(* CODESYS project comlibv2_gd.library
   Company: G.D Spa
   Version: 1.0.0.3
   Placeholder: COMlibV2_GD
   Title: COMlibV2_GD

Project tree, tasks and I/O mapping:
  libraries: Tc2_Standard, * (Beckhoff Automation GmbH); Tc2_System, * (Beckhoff Automation GmbH); Tc3_Module, * (Beckhoff Automation GmbH)
  Data types/
    COMlibV2/
      [Internal]/
        AdsSerialComm/
          data type ComADSSerialConfig_1
          data type ComADSServerCmd
        data type ComDebugBuffer
      AdsSerialComm/
        data type ComDTRCtrl_t
        data type ComRTSCtrl_t
        data type ComSerialConfig
        data type ComStopBits_t
      Hardware Types/
        data type EL6inData22B
        data type EL6outData22B
        data type IE6inData11B
        data type IE6outData11B
        data type KL6inData
        data type KL6inData22B
        data type KL6inData5B
        data type KL6outData
        data type KL6outData22B
        data type KL6outData5B
        data type M8000inData
        data type M8000outData
        data type PcComInData
        data type PcComOutData
      data type ComBuffer
      data type ComError_t
      data type ComHandshake_t
      data type ComParity_t
      data type ComRegisterData_t
      data type ComRegisterList_t
      data type ComSerialLineMode_t
  Global Variables/
    global variables Global_Constants
    global variables Global_Constants_ComLibVersion
    global variables Global_Variables
    global variables Variable_Configuration
  POUs/
    COMlibV2/
      [Internal]/
        function block _ReceiveString [ST]
        function block _SendString [ST]
        function _strncpy [ST]
      Background Communication/
        function block SerialLineControl [ST]
        function block SerialLineControlADS [ST]
        function block SerialLineControlM8000 [ST]
      CO_Nfiguration/
        function block KL6configuration [ST]
        function block KL6ReadRegisters [ST]
        function block KL6WriteRegisters [ST]
        function block M8000configuration [ST]
      Send + Receive/
        function block ReceiveByte [ST]
        function block ReceiveData [ST]
        function block ReceiveString [FBD]
        function block ReceiveString255 [FBD]
        function block SendByte [ST]
        function block SendData [ST]
        function block SendString [FBD]
        function block SendString255 [FBD]
      Version/
        function Get_ComLib_Version [ST]
      function ASC [ST]
      function CHR [ST]
      function block ClearComBuffer [ST]
      function block ComReset [ST]
  Version/
    global variables Global_Version
  Visualizations/
*)

// Data types/COMlibV2/[Internal]/AdsSerialComm/ComADSSerialConfig_1
{library private}
TYPE ComADSSerialConfig_1 :
(*	contains the configuration parameters of the com port to be opened.
	The same structure exists in the AdsSerialCommServer. *)
STRUCT
	StructVer	:UINT	:=1;	(* structure version *)									(* C++ -> unsigned __int16 *)
	TL			:UINT	:=0;	(* None=0;Error=1,Warning=2,Info=3,Verbose=4,Noise=5 *)	(* C++ -> unsigned __int16 *)

	Baudrate	:UDINT	:=9600;				(* baud rate *)								(* C++ -> unsigned __int32	-> dcb:BaudRate *)
	Parity		:INT	:=0;				(* [0=none;1=odd,2=even;3=mark;4=space] *)	(* C++ -> unsigned __int16	-> dcb:fParity & dcb:Parity *)
	DataBits	:INT	:=8;				(* [4; 5; 6; 7; 8] *)						(* C++ -> unsigned __int16	-> dcb:ByteSize *)
	StopBits	:INT	:=0;				(* [0=1; 1=1.5; 2=2] *)						(* C++ -> unsigned __int16	-> dcb:StopBits *)

	DTR			:INT	:=DTR_CTRL_HANDSHAKE;	(* 'Data Terminal Ready' signal *)		(* C++ -> unsigned __int16	-> dcb:fDtrControl *)
	RTS			:INT	:=RTS_CTRL_HANDSHAKE;	(* 'Request to Send' signal (=RFR) *)	(* C++ -> unsigned __int16	-> dcb:fRtsControl *)
	CTS_Out		:BOOL	:=FALSE;				(* 'Clear to Send' signal *)			(* C++ -> unsigned __int8	-> dcb:fOutxCtsFlow *)
	DSR_Out		:BOOL	:=FALSE;				(* 'Dataset Ready' signal *)			(* C++ -> unsigned __int8	-> dcb:fOutxDsrFlow *)
	DSR_Sens	:BOOL	:=FALSE;				(* 'Dataset Ready' signal *)			(* C++ -> unsigned __int8	-> dcb:fDsrSensitivity *)

	Reserved1	:BOOL;
	Reserved2	:INT;
END_STRUCT
END_TYPE

// Data types/COMlibV2/[Internal]/AdsSerialComm/ComADSServerCmd
{library private}
TYPE ComADSServerCmd :
(* the server commands are transmitted via Ads IdxOffset *)
(
	ASC_CMD_OPENPORT		:=1,
	ASC_CMD_CHECKPORT		:=2,
	ASC_CMD_CLOSEPORT		:=3,
	ASC_CMD_CHECKFORDATA	:=4,
	ASC_CMD_READDATA		:=5,
	ASC_CMD_WRITEDATA		:=6
);
END_TYPE

// Data types/COMlibV2/[Internal]/ComDebugBuffer
TYPE ComDebugBuffer :
STRUCT
	Buffer:	ARRAY[0..BUFFERSIZE_DEBUGBUFFER] OF INT;
	Status: 	ARRAY[0..BUFFERSIZE_DEBUGBUFFER] OF INT;
	Idx:		UINT;
END_STRUCT
END_TYPE

// Data types/COMlibV2/AdsSerialComm/ComDTRCtrl_t
TYPE ComDTRCtrl_t :
(
	DTR_CTRL_DISABLE,
	DTR_CTRL_ENABLE,
	DTR_CTRL_HANDSHAKE
);
END_TYPE

// Data types/COMlibV2/AdsSerialComm/ComRTSCtrl_t
TYPE ComRTSCtrl_t :
(
	RTS_CTRL_DISABLE,
	RTS_CTRL_ENABLE,
	RTS_CTRL_HANDSHAKE,
	RTS_CTRL_TOGGLE
);
END_TYPE

// Data types/COMlibV2/AdsSerialComm/ComSerialConfig
TYPE ComSerialConfig :
(* contains the configuration parameters of the com port to be opened. *)
STRUCT
	ComPort		:UDINT			:=1;					(* Serial port number [1..255] *)
	Baudrate	:UDINT			:=9600;
	Parity		:ComParity_t	:=PARITY_NONE;
	DataBits	:INT			:=8;					(* [4..8] *)
	StopBits	:ComStopBits_t	:=STOPBITS_ONE;

	DTR			:ComDTRCtrl_t	:=DTR_CTRL_HANDSHAKE;	(* 'Data Terminal Ready' signal *)
	RTS			:ComRTSCtrl_t	:=RTS_CTRL_HANDSHAKE;	(* 'Request to Send' signal (= RFR 'Ready for Receiving') *)
	CTS			:BOOL			:=FALSE;				(* 'Clear to Send' signal *)
	DSR			:BOOL			:=FALSE;				(* 'Dataset Ready' signal *)

	TraceLevel	:BYTE			:=0;					(* None=0;Error=1,Warning=2,Info=3,Verbose=4,Noise=5 *)

	Reserved1	:BYTE;
	Reserved2	:BYTE;
	Reserved3	:BYTE;
END_STRUCT
END_TYPE

// Data types/COMlibV2/AdsSerialComm/ComStopBits_t
TYPE ComStopBits_t :
(
	STOPBITS_ONE	:= 1,
	STOPBITS_TWO	:= 2,
	STOPBITS_ONE5	:= 3
);
END_TYPE

// Data types/COMlibV2/Hardware Types/EL6inData22B
(* This data type is corresponding to the
   KL-6xxx data structure used in the
   TwinCAT SystemManager
   (KL-6xxx version using 5 data bytes / 
    non-alternative (standard) output ) 
*)
TYPE EL6inData22B:
STRUCT
	Status: WORD;
	D: ARRAY[0..21] OF BYTE;
END_STRUCT
END_TYPE

// Data types/COMlibV2/Hardware Types/EL6outData22B
(* This data type is corresponding to the
   KL-6xxx data structure used in the
   TwinCAT SystemManager
   (KL-6xxx version using 5 data bytes / 
    non-alternative (standard) output ) 
*)
TYPE EL6outData22B:
STRUCT
	Ctrl: WORD;
	D: ARRAY[0..21] OF BYTE;
END_STRUCT
END_TYPE

// Data types/COMlibV2/Hardware Types/IE6inData11B
(* This data type is corresponding to the
   KL-6xxx data structure used in the
   TwinCAT SystemManager
   (KL-6xxx version using 5 data bytes / 
    non-alternative (standard) output ) 
*)
TYPE IE6inData11B:
STRUCT
	Status: BYTE;
	D: ARRAY[0..10] OF BYTE;
END_STRUCT
END_TYPE

// Data types/COMlibV2/Hardware Types/IE6outData11B
(* This data type is corresponding to the
   KL-6xxx data structure used in the
   TwinCAT SystemManager
   (KL-6xxx version using 5 data bytes / 
    non-alternative (standard) output ) 
*)
TYPE IE6outData11B:
STRUCT
	Ctrl: BYTE;
	D: ARRAY[0..10] OF BYTE;
END_STRUCT
END_TYPE

// Data types/COMlibV2/Hardware Types/KL6inData
(* This data type is corresponding to the
   KL-6xxx data structure used in the
   TwinCAT SystemManager
   (KL-6xxx version using 3 data bytes / alternative output)
*)
TYPE KL6inData:
STRUCT
	Status: BYTE;
	SerStatus: BYTE;
	D: ARRAY[0..2] OF BYTE;
END_STRUCT
END_TYPE

// Data types/COMlibV2/Hardware Types/KL6inData22B
(* This data type is corresponding to the
   KL-6xxx data structure used in the
   TwinCAT SystemManager
   (KL-6xxx version using 5 data bytes / 
    non-alternative (standard) output ) 
*)
TYPE KL6inData22B:
STRUCT
	Status: WORD;
	D: ARRAY[0..21] OF BYTE;
END_STRUCT
END_TYPE

// Data types/COMlibV2/Hardware Types/KL6inData5B
(* This data type is corresponding to the
   KL-6xxx data structure used in the
   TwinCAT SystemManager
   (KL-6xxx version using 5 data bytes / 
    non-alternative (standard) output ) 
*)
TYPE KL6inData5B:
STRUCT
	Status: BYTE;
	D: ARRAY[0..4] OF BYTE;
END_STRUCT
END_TYPE

// Data types/COMlibV2/Hardware Types/KL6outData
(* This data type is corresponding to the
   KL-6xxx data structure used in the
   TwinCAT SystemManager
   (KL-6xxx version using 3 data bytes / alternative output)
*)
TYPE KL6outData:
STRUCT
	Ctrl: BYTE;
	SerCtrl: BYTE;
	D: ARRAY[0..2] OF BYTE;
END_STRUCT
END_TYPE

// Data types/COMlibV2/Hardware Types/KL6outData22B
(* This data type is corresponding to the
   KL-6xxx data structure used in the
   TwinCAT SystemManager
   (KL-6xxx version using 5 data bytes / 
    non-alternative (standard) output ) 
*)
TYPE KL6outData22B:
STRUCT
	Ctrl: WORD;
	D: ARRAY[0..21] OF BYTE;
END_STRUCT
END_TYPE

// Data types/COMlibV2/Hardware Types/KL6outData5B
(* This data type is corresponding to the
   KL-6xxx data structure used in the
   TwinCAT SystemManager
   (KL-6xxx version using 5 data bytes / 
    non-alternative (standard) output ) 
*)
TYPE KL6outData5B:
STRUCT
	Ctrl: BYTE;
	D: ARRAY[0..4] OF BYTE;
END_STRUCT
END_TYPE

// Data types/COMlibV2/Hardware Types/M8000inData
(* This data type is corresponding to the
   KL-6xxx data structure used in the
   TwinCAT SystemManager
   (KL-6xxx version using 3 data bytes / alternative output)
*)
TYPE M8000inData:
STRUCT
	D: ARRAY[0..3] OF BYTE;
END_STRUCT
END_TYPE

// Data types/COMlibV2/Hardware Types/M8000outData
(* This data type is corresponding to the
   KL-6xxx data structure used in the
   TwinCAT SystemManager
   (KL-6xxx version using 3 data bytes / alternative output)
*)
TYPE M8000outData:
STRUCT
	D: ARRAY[0..3] OF BYTE;
END_STRUCT
END_TYPE

// Data types/COMlibV2/Hardware Types/PcComInData
(* This data type is corresponding to the
   PC COM-Port data structure used in
   the TwinCAT SystemManager. 
   (KL-6xxx emulation mode with 64 data bytes)
*)
TYPE PcComInData:
STRUCT
	SerStatus: WORD;
	D: ARRAY[0..63] OF BYTE;
END_STRUCT
END_TYPE

// Data types/COMlibV2/Hardware Types/PcComOutData
(* This data type is corresponding to the
   PC COM-Port data structure used in
   the TwinCAT SystemManager. 
   (KL-6xxx emulation mode with 64 data bytes)
*)
TYPE PcComOutData:
STRUCT
	SerCtrl: WORD;
	D: ARRAY[0..63] OF BYTE;
END_STRUCT
END_TYPE

// Data types/COMlibV2/ComBuffer
(* This data type will be used as a software character buffer
   between serial line I/O and user functions as ReceiveByte
   or SendByte.
*)
TYPE ComBuffer:
STRUCT
	Buffer:	ARRAY[0..1028] OF BYTE;	(* ringbuffer *)
	RdIdx:	UINT;		(* first valid byte in ringbuffer *)
	WrIdx:	UINT;		(* first invalid byte in ringbuffer *)
	Count:	UINT;		(* number of bytes in ringbuffer *)
	FreeByte:UINT;		(* number of free bytes in ringbuffer *)
	Error:	UINT;		(* error code of serial line interface *)
	blocked	: BOOL;		(* semaphore for task synchronization *)
END_STRUCT
END_TYPE

// Data types/COMlibV2/ComError_t
TYPE ComError_t :
 (
	COMERROR_NOERROR 				:= 0,
	COMERROR_PARAMETERCHANGED		:= 1,		(* input parameters changed during reception *)
	COMERROR_TXBUFFOVERRUN			:= 2,		(* string > transmit buffer *)
	COMERROR_STRINGOVERRUN			:= 10,		(* end of string *)
	COMERROR_ZEROCHARINVALID 		:= 11,		(* string cannot receive zero characters *)
	COMERROR_INVALIDPOINTER			:= 20,		(* invalid data pointer, e. g. zero *)
	COMERROR_INVALIDRXPOINTER		:= 21,		(* invalid data pointer for ReceiveData *)
	COMERROR_INVALIDRXLENGTH 		:= 22,		(* invalid length for ReceiveData, e. g. zero *)
	COMERROR_DATASIZEOVERRUN 		:= 23,		(* end of data block *)
	COMERROR_INVALIDPROCESSDATASIZE	:= 24,
	COMERROR_MODENOTSUPPORTED		:= 16#0101,	(* mode not supported (3-Byte Terminals connectd to bus controllers) *)
	COMERROR_INVALIDCHANNELNUMBER	:= 16#0102,
	COMERROR_INVALIDBAUDRATE 		:= 16#1001,
	COMERROR_INVALIDNUMDATABITS		:= 16#1002,
	COMERROR_INVALIDNUMSTOPBITS		:= 16#1003,
	COMERROR_INVALIDPARITY			:= 16#1004,
	COMERROR_INVALIDHANDSHAKE		:= 16#1005,
	COMERROR_INVALIDNUMREGISTERS	:= 16#1006,
	COMERROR_INVALIDREGISTER		:= 16#1007,
	COMERROR_TIMEOUT				:= 16#1008
 );
END_TYPE

// Data types/COMlibV2/ComHandshake_t
TYPE ComHandshake_t :
 (
	HANDSHAKE_NONE,
	HANDSHAKE_RTSCTS,
	HANDSHAKE_XONXOFF,
	RS485_FULLDUPLEX,
	RS485_HALFDUPLEX,
	RS485_FULLDUPLEX_XONXOFF,
	RS485_HALFDUPLEX_XONXOFF
 );
END_TYPE

// Data types/COMlibV2/ComParity_t
TYPE ComParity_t :
 (
	PARITY_NONE,
	PARITY_EVEN,
	PARITY_ODD,
	PARITY_MARK,	(* only available with SerialLineControlADS *)
	PARITY_SPACE	(* only available with SerialLineControlADS *)
 );
END_TYPE

// Data types/COMlibV2/ComRegisterData_t
TYPE ComRegisterData_t :
STRUCT
	Register : BYTE;
	Value : WORD;
END_STRUCT
END_TYPE

// Data types/COMlibV2/ComRegisterList_t
TYPE ComRegisterList_t : ARRAY[0..63] OF ComRegisterData_t;
END_TYPE

// Data types/COMlibV2/ComSerialLineMode_t
TYPE ComSerialLineMode_t :
 (
 	SERIALLINEMODE_DEFAULT,
 	SERIALLINEMODE_KL6_3B_ALTERNATIVE,
 	SERIALLINEMODE_KL6_5B_STANDARD,
 	SERIALLINEMODE_KL6_22B_STANDARD,
 	SERIALLINEMODE_PC_COM_PORT,
 	SERIALLINEMODE_EL6_22B,
 	SERIALLINEMODE_IE6_11B
 );
END_TYPE

// Global Variables/Global_Constants
{attribute 'Tc2GvlVarNames'}
VAR_GLOBAL CONSTANT
(* constants for error codes returned as nErrorID output of SerialLineControlADS *)
	(* invalid input parameters *)
	COMERRORADS_INVALID_COMPORT		:UDINT:=16#00009001;
	COMERRORADS_INVALID_CMD			:UDINT:=16#00009002;
	COMERRORADS_INVALID_DATAPOINTER	:UDINT:=16#00009003;
	COMERRORADS_INVALID_CFGSTLEN	:UDINT:=16#00009011;
	COMERRORADS_INVALID_CFGSTVER	:UDINT:=16#00009012;	(* unknown configuration structure version *)
	COMERRORADS_INVALID_TL			:UDINT:=16#00009013;	(* invalid TraceLevel *)
	COMERRORADS_INVALID_BAUDRATE	:UDINT:=16#00009021;
	COMERRORADS_INVALID_PARITY		:UDINT:=16#00009022;
	COMERRORADS_INVALID_DATABITS	:UDINT:=16#00009023;
	COMERRORADS_INVALID_STOPBITS	:UDINT:=16#00009024;
	COMERRORADS_INVALID_DTR_CTRL	:UDINT:=16#00009025;
	COMERRORADS_INVALID_RTS_CTRL	:UDINT:=16#00009026;
	COMERRORADS_INVALID_CTS_OUTCTRL	:UDINT:=16#00009027;
	COMERRORADS_INVALID_DSR_OUTCTRL	:UDINT:=16#00009028;
	COMERRORADS_INVALID_DSR_SENS	:UDINT:=16#00009029;
	(* Specific Error Codes *)
	COMERRORADS_NOT_INIT			:UDINT:=16#00009031;
	COMERRORADS_RD_BUFFER_OVERRUN	:UDINT:=16#00009032;
	COMERRORADS_PORT_CONNECTED		:UDINT:=16#00009033;	(* port already opened by the server *)
	COMERRORADS_PORT_NOT_CONNECTED	:UDINT:=16#00009034;	(* port not yet opened by the server *)
	COMERRORADS_RD_THREAD_TIMEOUT	:UDINT:=16#00009035;
	COMERRORADS_WR_THREAD_TIMEOUT	:UDINT:=16#00009036;
	COMERRORADS_RD_FAILURE			:UDINT:=16#00009037;
	COMERRORADS_WR_FAILURE			:UDINT:=16#00009038;
	(* error codes out of Plc library *)
	COMERRORADS_SERVER_INCOMPATIBLE	:UDINT:=16#00009101;	(* server version incompatible *)

{library private}
	BUFFERSIZE_DEBUGBUFFER : INT:= 300;
{library public}
END_VAR

// Global Variables/Global_Constants_ComLibVersion
{attribute 'Tc2GvlVarNames'}
VAR_GLOBAL CONSTANT
	VERSION_COMLIB : STRING(20) := '2.003.008';
END_VAR

// Global Variables/Global_Variables
{attribute 'Tc2GvlVarNames'}
VAR_GLOBAL
END_VAR

// Global Variables/Variable_Configuration
{attribute 'Tc2GvlVarNames'}
VAR_CONFIG
END_VAR

// Version/Global_Version
{attribute 'TcGenerated'}
// This function has been automatically generated from the project information.
VAR_GLOBAL CONSTANT
	{attribute 'const_non_replaced'}
	{attribute 'linkalways'}
	stLibVersion_COMlibV2_GD : ST_LibVersion := (iMajor := 1, iMinor := 0, iBuild := 0, iRevision := 3, sVersion := '1.0.0.3');
END_VAR

// POUs/COMlibV2/[Internal]/_ReceiveString
FUNCTION_BLOCK _ReceiveString
VAR_INPUT
	Prefix : STRING;
	Suffix : STRING;
	Timeout: TIME;
	Reset  : BOOL;
	pReceivedString : POINTER TO BYTE;	(* Pointer to variable length string *)
	SizeReceivedString : INT;	(* variable string size *)
END_VAR
VAR_OUTPUT
	StringReceived:	BOOL;
	Busy :			BOOL;
	Error:			ComError_t;
	RxTimeout : 	BOOL;
	ErrorCountPrefix : INT; (* invalid characters received before prefix *)
	ReceivedPrefix : STRING;(* received prefix including invalid characters *)
END_VAR
VAR_IN_OUT
	RXbuffer :		COMbuffer;
END_VAR
VAR
	RxString : STRING(255);
	state: INT;
	c : BYTE;
	l : INT;
	l2 : INT;
	pl : INT;
	sl : INT;
	iTimeout : TIME;
	Receive : ReceiveByte;
	TimeoutTimer : TOF;
END_VAR

IF Reset THEN
	state := 0;
	RETURN;
END_IF

IF state = 0 THEN
	StringReceived := FALSE;
	busy := FALSE;
	Error := 0;
	RxTimeout := FALSE;
	RxString := '';
	l := 0;
	state := 1;
ELSE
	REPEAT
		(* receive one character *)
		Receive(RXbuffer:=RXbuffer);

		TimeoutTimer( IN:=Receive.ByteReceived, PT:=iTimeout );

		IF  Receive.ByteReceived THEN
			c := Receive.ReceivedByte;
			IF c = 0 THEN (* 20.11.2000, KSt *)
				Error := COMERROR_ZEROCHARINVALID;
				busy := FALSE;
				state := 0;
			ELSE
				IF state = 1 THEN
					busy := TRUE;
					l := 0;
					ErrorCountPrefix := 0;
					ReceivedPrefix := '';
					pl := LEN(Prefix);
					sl := LEN(Suffix);
					iTimeout := Timeout;
					IF sl = 0 AND iTimeout = T#0s THEN (* 2.1.2002, KSt, Reihenfolge umgestellt *)
						iTimeout := T#1s;
					END_IF
					IF pl > 0 THEN
						state := 10;
					ELSE
						state := 20;
					END_IF
				END_IF

				CASE state OF
					10 :	(* Wait for prefix *)
						RxString := CONCAT(RxString, CHR(c) );
						ReceivedPrefix := CONCAT(ReceivedPrefix, CHR(c) );
						l2 := LEN(RxString);
						IF (l >= l2) OR (l2>=SizeReceivedString) THEN
							(* stringsize reached *)
							Error := COMERROR_STRINGOVERRUN;
							(* pReceivedString^ := LEFT(RxString,SizeReceivedString-1);*)
							_strncpy(pTargetString:=pReceivedString, pSourceString:=ADR(RxString), MaxSize:=SizeReceivedString); (* 3.6.2002 KST *)
							StringReceived := TRUE;
							busy := FALSE;
							state := 0;
						ELSE
							l := l2;
							IF l <= pl THEN
								IF LEFT(Prefix, l) <> RxString THEN
									RxString := '';
									ErrorCountPrefix := ErrorCountPrefix + 1;
									l := 0;
								ELSE
									IF l = pl THEN
										state := 20;
									END_IF
								END_IF
							END_IF
						END_IF

					20 :	(* Wait for suffix *)
						RxString := CONCAT(RxString, CHR(c) );
						l2 := LEN(RxString);
						IF (l >= l2) OR (l2>=SizeReceivedString) THEN
							(* stringsize reached *)
							Error := COMERROR_STRINGOVERRUN;
							(* pReceivedString^ := LEFT(RxString,SizeReceivedString-1); *)
							_strncpy(pTargetString:=pReceivedString, pSourceString:=ADR(RxString), MaxSize:=SizeReceivedString); (* 3.6.2002 KST *)
							StringReceived := TRUE;
							busy := FALSE;
							state := 0;
						ELSE
							l := l2;
							IF (sl > 0) AND (l >= pl + sl) THEN
								IF RIGHT(RxString, sl) = Suffix THEN
									(* pReceivedString^ := RxString; *)
									_strncpy(pTargetString:=pReceivedString, pSourceString:=ADR(RxString), MaxSize:=SizeReceivedString); (* 3.6.2002 KST *)
									StringReceived := TRUE;
									busy := FALSE;
									state := 0;
								END_IF
							END_IF
						END_IF
				END_CASE
			END_IF
		ELSE
			(* no char received *)
			IF state > 1 AND l > 0 AND iTimeout > T#0s AND NOT TimeoutTimer.Q THEN
				(* pReceivedString^ := RxString; *)
				_strncpy(pTargetString:=pReceivedString, pSourceString:=ADR(RxString), MaxSize:=SizeReceivedString); (* 3.6.2002 KST *)
				StringReceived := TRUE;
				busy := FALSE;
				RxTimeout := TRUE;
				state := 0;
			END_IF
			(* check if input parameters have changed, 30.12.2002 KSt *)
			IF state > 1 AND (pl<>LEN(Prefix) OR sl<>LEN(Suffix) OR iTimeout<>Timeout) THEN
				Error := COMERROR_PARAMETERCHANGED;
				busy := FALSE;
				state := 0;
			END_IF
		END_IF
	UNTIL NOT busy OR NOT Receive.ByteReceived
	END_REPEAT
END_IF

END_FUNCTION_BLOCK

// POUs/COMlibV2/CHR
FUNCTION CHR : STRING
VAR_INPUT
	c : BYTE;
END_VAR
VAR
	str1: STRING(1);
	pChar : POINTER TO BYTE;
END_VAR

	str1 := '@'; (* initialization with any character *)
	pChar := ADR(str1);	(* get string pointer *)
	pChar^ := c; (* overwrite first character with c *)
	CHR := str1; (* return c as string *)

END_FUNCTION

// POUs/COMlibV2/[Internal]/_strncpy
FUNCTION _strncpy : BOOL
VAR_INPUT
	pTargetString 	: POINTER TO BYTE;
	pSourceString	: POINTER TO BYTE;
	MaxSize 			: INT;
END_VAR
VAR
	d 	: XWORD;
	i	: INT;
END_VAR

FOR i := 1 TO MaxSize-1 DO
	pTargetString^ := pSourceString^;
	d := pTargetString;
	d := d + 1;
	pTargetString := d;
	d := pSourceString;
	d := d + 1;
	pSourceString := d;

(*	vorzeitiger Abbruch des Loops ist leider nicht moeglich,
	weil auch die Zeichen nach der teminierenden Null im 
	debug-Fenster angezeigt werden.
*)
(*	IF pSourcestring^ = 0 THEN	*)
(*		EXIT; 	 (for loop) 	*)
(*	END_IF						*)
END_FOR
(* pTargetString := 0; *)	(* 2011-01-12 KSt nach Meldung von Dieter Auer *)
pTargetString^ := 0;	(* 2011-01-12 KSt nach Meldung von Dieter Auer *)

END_FUNCTION

// POUs/COMlibV2/Send + Receive/ReceiveByte
(*=================================================================
 *	
 *	Modul:	ReceiveByte
 *			The function block reads one byte out of
 * 			the software buffer (ComBuffer) if available.
 *	Date: 	11.8.98
 *
 *=================================================================
 *)
FUNCTION_BLOCK ReceiveByte
VAR_OUTPUT
	ByteReceived:	BOOL;
	ReceivedByte:	BYTE;
	Error:			ComError_t;
END_VAR
VAR_IN_OUT
	RxBuffer :		COMbuffer;
END_VAR
VAR
END_VAR

	Error := RXbuffer.Error;
	IF Error <> COMERROR_NOERROR THEN
		RETURN;
	END_IF

	IF RXbuffer.Count > 0 THEN
		RXbuffer.blocked := TRUE;	(* block fast PLC Task *)
		ReceivedByte :=RXbuffer.Buffer[RXbuffer.RdIdx];
		RXbuffer.RdIdx := RXbuffer.RdIdx + 1;
		IF RXbuffer.RdIdx >= SIZEOF(RxBuffer.Buffer)  THEN
			RXbuffer.RdIdx := 0;
		END_IF
		RXbuffer.Count := RXbuffer.Count -1;
		RXbuffer.FreeByte :=SIZEOF(RxBuffer.Buffer) - RXbuffer.Count;
		ByteReceived := TRUE;
		RXbuffer.blocked := FALSE;	(* unblock fast PLC Task *)
	ELSE
		ByteReceived := FALSE;
		ReceivedByte := 0;
	END_IF

END_FUNCTION_BLOCK

// POUs/COMlibV2/[Internal]/_SendString
FUNCTION_BLOCK _SendString
VAR_INPUT
	SendString:	STRING(255);
END_VAR
VAR_OUTPUT
	Busy : 		BOOL;
	Error:		ComError_t;
END_VAR
VAR_IN_OUT
	TXbuffer:	COMbuffer;
END_VAR
VAR
	pos : INT;
	Send : SendByte;
	c : BYTE;
	ls: INT;
END_VAR

 	IF NOT Busy THEN
		pos := 1;
		Busy := TRUE;
	END_IF

	IF Send.Busy THEN
		Send( TxBuffer := TxBuffer );
		Error := Send.Error; (* 2011-06-24 JANZ: line added because otherwise in case of buffer overrun at last byte: error keeps at output although it was sent successfully. *)
	ELSE
		ls :=LEN(SendString); (* moved out of the repeat loop - 20080520 KSt *)
		REPEAT
(*			IF NOT Send.Busy OR Send.Error = COMERROR_TXBUFFOVERRUN THEN *) (* 2011-06-24 JANZ if condition removed because line is needless (Send.Busy always FALSE here) *)
				IF pos > ls THEN
					busy := FALSE;
				ELSE
					c := ASC(MID( SendString, 1, pos ));
					Send( SendByte := c, TxBuffer := TxBuffer );
					Error := Send.Error;
(*					IF Send.Error = 0 THEN	*)	(* 2010-02-19 KSt IF condition removed *)
					pos := pos + 1;
(*					END_IF;	*)					(* 2010-02-19 KSt IF condition removed *)
				END_IF
(*			END_IF *)							(* 2011-06-24 JANZ if condition removed *)
		UNTIL Send.Busy OR NOT busy
		END_REPEAT
	END_IF

END_FUNCTION_BLOCK

// POUs/COMlibV2/Send + Receive/SendString
FUNCTION_BLOCK SendString
VAR_INPUT
	SendString:	STRING;
END_VAR
VAR_OUTPUT
	Busy : 		BOOL;
	Error:		ComError_t;
END_VAR
VAR_IN_OUT
	TXbuffer:	COMbuffer;
END_VAR
VAR
END_VAR
VAR
	SendStringStandard: _SendString;
END_VAR

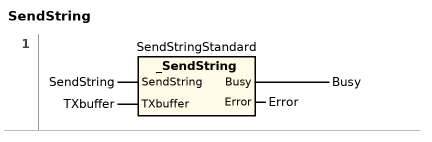
// NETWORK 1
SendStringStandard(SendString := SendString, TXbuffer := TXbuffer, Error => Error); // _SendString
Busy := SendStringStandard.Busy;

END_FUNCTION_BLOCK

// POUs/COMlibV2/ASC
FUNCTION ASC : BYTE
VAR_INPUT
	str : STRING;
END_VAR
VAR
	pChar : POINTER TO BYTE;
END_VAR

	pChar := ADR(str);
	ASC := pChar^;

END_FUNCTION

// POUs/COMlibV2/Send + Receive/SendByte
(*=================================================================
 *
 *	Modul:	SendByte
 *			The function block writes one byte into
 * 			the software buffer (ComBuffer).
 *	Date: 	11.8.98
 *
 *=================================================================
 *)
FUNCTION_BLOCK SendByte
VAR_INPUT
	SendByte:	BYTE;
END_VAR
VAR_OUTPUT
	Busy : 		BOOL;
	Error:		ComError_t;
END_VAR
VAR_IN_OUT
	TxBuffer:	COMbuffer;
END_VAR
VAR
END_VAR

	Busy := TRUE;
	Error := TXbuffer.Error;
	IF Error <> COMERROR_NOERROR THEN
		RETURN;
	END_IF

	TXbuffer.FreeByte := SIZEOF(TxBuffer.Buffer) - TXbuffer.Count;
	IF TXbuffer.FreeByte > 1 THEN
		TXbuffer.blocked := TRUE;	(* block fast PLC Task *)
		TXbuffer.Buffer[TXbuffer.WrIdx] := SendByte;
		TXbuffer.WrIdx := TXbuffer.WrIdx + 1;
		IF TXbuffer.WrIdx >= SIZEOF(TxBuffer.Buffer)  THEN
			TXbuffer.WrIdx := 0;
		END_IF
		TXbuffer.Count := TXbuffer.Count + 1;
		TXbuffer.FreeByte := SIZEOF(TxBuffer.Buffer) - TXbuffer.Count;
		Busy := FALSE;
		TXbuffer.blocked := FALSE;	(* unblock fast PLC Task *)
	ELSE
		Error := COMERROR_TXBUFFOVERRUN;
	END_IF

END_FUNCTION_BLOCK

// POUs/COMlibV2/Background Communication/SerialLineControl
(* =============================================================
 *	Modul:	Serial line interface controller for background communication
 *			supports multiple interface types like 
 *			KL6xxx 3 byte alternative mode
 *			KL6xxx 5 byte standard mode
 *			KL6xxx 22 byte standard mode with extended process data interface
 *			KL6xxx 64 byte PC COM port
 *			EL6xxx 22 byte 
 *			IP6xxx 11 byte
 *			communication between a serial line hardware device and 
 *			PLC communication buffers (RxBuffer, TxBuffer)
 *
 *	Date: 	21.12.2004
 * ============================================================= *)
FUNCTION_BLOCK SerialLineControl
VAR_INPUT
	Mode		:ComSerialLineMode_t;
	pComIn		:POINTER TO ARRAY[0..65] OF BYTE; (* must meet the maximum size of a hardware related data structure *)
	pComOut		:POINTER TO ARRAY[0..65] OF BYTE; (* must meet the maximum size of a hardware related data structure *)
	SizeComIn	:INT;
END_VAR
VAR_OUTPUT
	Error		:BOOL;
	ErrorID		:ComError_t;
END_VAR
VAR_IN_OUT
	TxBuffer	:COMbuffer;
	RxBuffer	:COMbuffer;
END_VAR
VAR
	ComPortDebugBuffer:ComDebugBuffer;
	InvalidDataExchangeMode: UINT;
	RegisterMode: UINT;
	pCTRL: POINTER TO WORD;
	pSTATUS: POINTER TO WORD;
	RxCount: WORD;
	TxCount: WORD;
	DataIndex: UINT;
	DataCountMask: WORD;
	DataCountShift: BYTE;
	ReceiveHandshakeBit :	WORD;
	TransmitHandshakeBit : 	WORD;
	TransmitBufferSentBit: WORD;
	ContinousModeStartBit : WORD;
	ReceiveBufferFullBit: WORD;
	ResetBit: WORD;
	RR: WORD;
	RA: WORD;
	TR: WORD;
	TA: WORD;
	IA: WORD;
	BUF_F: WORD;
	noTAcounter: BYTE;
	initialized: BOOL;
	TransmitDataSent: BOOL;
	i: UINT;
END_VAR

IF pComIn=0 OR pComOut=0 OR SizeComIn=0 THEN
	Error := TRUE;
	ErrorID := COMERROR_INVALIDPOINTER;
	RETURN;
ELSIF SizeComIn<>5 AND Mode=SERIALLINEMODE_KL6_3B_ALTERNATIVE THEN
	Error := TRUE;
	ErrorID := COMERROR_MODENOTSUPPORTED; (* 3 byte terminal connected to bus controllers *)
	RETURN;
ELSE
	Error := FALSE;
	ErrorID := 0;
END_IF

pCTRL := pComOut;
pSTATUS := pComIn;
InvalidDataExchangeMode := 	(pCTRL^ 	AND 2#00000000_10000100) OR	(* register mode or initialization *)
							(pSTATUS^	AND 2#00000000_10000000);	(* register mode or initialization *)
RegisterMode := 				(pCTRL^ 	AND 2#00000000_10000000) OR	(* register mode *)
							(pSTATUS^	AND 2#00000000_10000000);	(* register mode *)
ReceiveHandshakeBit 	:= 2#00000000_00000010;	(* RA / RR *)
TransmitHandshakeBit := 2#00000000_00000001;	(* TA / TR *)
ResetBit			 	:= 2#00000000_00000100;	(* IA *)
TransmitBufferSentBit 	:= 2#00000000_00000100;	(* same as IA bit - double function *)
ContinousModeStartBit 	:= 2#00000000_00001000;
ReceiveBufferFullBit	:= 2#00000000_00001000;	(* BUF_F *)
DataIndex := 2; (* array index after control and serial control *)

IF SizeComIn = 5 THEN
	(* 3 byte alternative mode *)
	InvalidDataExchangeMode := 	(pCTRL^ 	AND 2#00000100_10000000) OR	(* register mode or initialization *)
								(pSTATUS^	AND 2#00000000_10000000);	(* register mode or initialization *)
	RegisterMode := 				(pCTRL^ 	AND 2#00000000_10000000) OR	(* register mode *)
								(pSTATUS^	AND 2#00000000_10000000);	(* register mode *)
	DataCountMask 		:= 2#01110000_00000000;
	DataCountShift := 12;
	ReceiveHandshakeBit 	:= 2#00000010_00000000;	(* RA / RR *)
	TransmitHandshakeBit	:= 2#00000001_00000000;	(* TA / TR *)
	ResetBit			 	:= 2#00000100_00000000;	(* IA / IR *)
	TransmitBufferSentBit	:= 2#00000100_00000000; 	(* same as IA bit - double function *)
	ContinousModeStartBit 	:= 2#00001000_00000000;
	ReceiveBufferFullBit	:= 2#00001000_00000000;	(* BUF_F *)
ELSIF SizeComIn = 12 AND Mode=SERIALLINEMODE_IE6_11B THEN
	(* IP6002-0001 with 11 data bytes plus status *)
	ReceiveBufferFullBit := 0; (* not supported *)
	DataIndex := 1; (* after 1 byte control *)
	DataCountMask := 2#00000000_01111000;
	DataCountShift := 3;
ELSIF SizeComIn < 8 THEN
	(* KL6 in standard mode - up to 7 bytes *)
	DataIndex := 1; (* after 1 byte control *)
	DataCountMask := 2#00000000_01110000;
	DataCountShift := 4;
ELSIF SizeComIn >= 66 THEN
	(* PC COM port *)
	DataCountMask := 2#11111111_11110000;
	DataCountShift := 4;
	InvalidDataExchangeMode := 0;
	RegisterMode := 0;
ELSE
	(* KL6 long data size - more than 7 bytes (22 byte) *)
	DataCountMask := 2#11111111_00000000;
	DataCountShift := 8;
END_IF

IF initialized THEN
	IF  InvalidDataExchangeMode = 0 THEN (* don't talk to the terminal during reset or register access *)

		(* Read data from serial interface to RxBuffer *)
		IF NOT RXbuffer.blocked THEN (* check if the buffer is blocked by the standard PLC task *)
			RxCount := SHR( pSTATUS^ AND DataCountMask, DataCountShift );
			RA := pCTRL^ AND ReceiveHandshakeBit;
			RR := pSTATUS^ AND ReceiveHandshakeBit;
			RXbuffer.FreeByte := SIZEOF(RXbuffer.Buffer) - RXbuffer.Count;
			IF RA<>RR AND RxCount <= RxBuffer.FreeByte THEN
				FOR i := 0 TO RxCount-1 DO
					(* copy data byte from the I/O buffer *)
					RXbuffer.Buffer[RXbuffer.WrIdx] := pComIn^[DataIndex+i];
					RXbuffer.WrIdx := RXbuffer.WrIdx + 1;
					IF RXbuffer.WrIdx >= SIZEOF(RXbuffer.Buffer) THEN
						RXbuffer.WrIdx := 0;
					END_IF
					(* copy data byte the the debug buffer *)
					ComPortDebugBuffer.Buffer[ComPortDebugBuffer.Idx]:=BYTE_TO_INT(pComIn^[DataIndex+i]);
					ComPortDebugBuffer.Status[ComPortDebugBuffer.Idx]:=1;
					IF UINT_TO_INT(ComPortDebugBuffer.Idx) < BUFFERSIZE_DEBUGBUFFER THEN
						ComPortDebugBuffer.Idx := ComPortDebugBuffer.Idx + 1;
					ELSE
						ComPortDebugBuffer.Idx:=0;
					END_IF
				END_FOR
				RXbuffer.Count := RXbuffer.Count + RxCount;
				RXbuffer.FreeByte := SIZEOF(RXbuffer.Buffer) - RXbuffer.Count;
				pCTRL^ := pCTRL^ XOR ReceiveHandshakeBit;	(* confirm *)
			END_IF
		END_IF

		(* Write data TxBuffer to serial interface *)
		IF NOT TXbuffer.blocked THEN
			IA := pSTATUS^ AND TransmitBufferSentBit;
			IF TxBuffer.Count > 0 THEN (* check if the buffer is blocked by the standard PLC task *)
				TA := pSTATUS^ AND TransmitHandshakeBit;
				TR := pCTRL^ AND TransmitHandshakeBit;
				BUF_F := pSTATUS^ AND ReceiveBufferFullBit;
				IF TA<>TR THEN (* if transmit dat not accepted *)
					noTAcounter := noTAcounter + 1;
					IF (noTAcounter >= 3) AND (IA=0) THEN
						(* if transmit dat not accepted for at least 3 cycles and transmit buffer is not empty *)
						pCTRL^ := pCTRL^ OR ContinousModeStartBit;	(* start continous transmission *)
					END_IF
				ELSE
					noTAcounter := 0; (* reset counter *)
					TxCount := INT_TO_WORD(SizeComIn) - UINT_TO_WORD(DataIndex);
					IF TxCount > TxBuffer.Count THEN
						TxCount := TxBuffer.Count;
					END_IF
					FOR i := 0 TO TxCount-1 DO
						(* copy data byte to the I/O buffer *)
						pComOut^[DataIndex+i] := TxBuffer.Buffer[TXbuffer.RdIdx];
						TXbuffer.RdIdx := TXbuffer.RdIdx + 1;
						IF TXbuffer.RdIdx >= SIZEOF(TXbuffer.Buffer) THEN
							TXbuffer.RdIdx := 0;
						END_IF
						(* copy data byte the the debug buffer *)
						ComPortDebugBuffer.Buffer[ComPortDebugBuffer.Idx]:=BYTE_TO_INT(pComOut^[DataIndex+i]);
						ComPortDebugBuffer.Status[ComPortDebugBuffer.Idx]:=2;
						IF UINT_TO_INT(ComPortDebugBuffer.Idx) < BUFFERSIZE_DEBUGBUFFER THEN
							ComPortDebugBuffer.Idx := ComPortDebugBuffer.Idx + 1;
						ELSE
							ComPortDebugBuffer.Idx:=0;
						END_IF
					END_FOR
					TXbuffer.Count := TXbuffer.Count - TxCount;
					TXbuffer.FreeByte := SIZEOF(TXbuffer.Buffer) - TXbuffer.Count;
					pCTRL^ := pCTRL^ AND NOT DataCountMask;
					pCTRL^ := pCTRL^ OR SHL( TxCount, DataCountShift);
(* 18.10.2005 - kein Zurücksetzen des ContinousModeStart bits, da sonst unnoetige Pause solange noch weitere Daten anstehen *)
(*					IF IA <> 0 THEN *)(* if transmit buffer sent *)
(* 						pCTRL^ := pCTRL^ AND NOT ContinousModeStartBit;*)	(* clear continous transmission *)
(*					END_IF*)
					pCTRL^ := pCTRL^ XOR TransmitHandshakeBit;	(* request *)
					TransmitDataSent := TRUE;
				END_IF
			ELSE (* no data to send *)
				IF TransmitDataSent THEN
					pCTRL^ := pCTRL^ OR ContinousModeStartBit;	(* start continous transmission *)
					TransmitDataSent := FALSE;
				ELSIF IA <> 0 THEN (* if transmit buffer sent *)
					pCTRL^ := pCTRL^ AND NOT ContinousModeStartBit;	(* clear continous transmission *)
				END_IF
			END_IF
		END_IF
	END_IF

ELSIF RegisterMode = 0 THEN
	(* initialization *)
	IF i = 0 THEN
		pCTRL^ := ResetBit;	(* request IR *)
	END_IF
	IA := pSTATUS^ AND ResetBit;
	IF IA <> 0 THEN
		pCTRL^ := 0;
		i := 1;
	ELSIF i=1 THEN
		initialized := TRUE;
	END_IF
END_IF

END_FUNCTION_BLOCK

// POUs/COMlibV2/Background Communication/SerialLineControlADS
(*=====================================================================================================*
 * Serial line interface controller for background communication                                       *
 * supports Pc ComPorts or Virtual ComPorts at the local PC or any connected PC (via Ads)              *
 * where TwinCAT TcAdsSerialCommServer is started. Communication is handled over ADS via Server.       *
 * Communication between a TwinCAT TcAdsSerialCommServer and                                           *
 * PLC communication buffers (RxBuffer, TxBuffer).                                                     *
 *=====================================================================================================*)
FUNCTION_BLOCK SerialLineControlADS
VAR_INPUT
	Connect		:BOOL;						(* connect to serial port [TRUE=connect, FALSE=disconnect] *)
	SerialCfg	:ComSerialConfig;
	NetId		:T_AmsNetId :='';			(* host NetId *)
	Timeout		:TIME :=DEFAULT_ADS_TIMEOUT;(* Timeout for ADS calls *)
END_VAR
VAR_IN_OUT
	TxBuffer    :ComBuffer;         (* serial Tx ComBuffer *)
	RxBuffer    :ComBuffer;         (* serial Rx ComBuffer *)
END_VAR
VAR_OUTPUT
	PortOpened	:BOOL;				(* Indicates if selected serial port is opened *)
	Error		:BOOL;				(* 'TRUE' if an error occurred *)
	ErrorID		:UDINT;				(* Displays the error code; 0 = no error *)
	Busy		:BOOL;				(* 'TRUE' if internal ADS communication is busy *)
	TxBufCount	:UDINT;				(* number of bytes in internal Tx buffer *)
	RxBufCount	:UDINT;				(* number of bytes in internal Rx buffer *)
END_VAR
{library private}
VAR
	NetId_Act		:T_AmsNetId := 'invalid';	(* initialized with invalid NetId to force INIT state *)
	Timeout_Act		:TIME :=DEFAULT_ADS_TIMEOUT;(* Timeout for ADS calls *)
	SerialCfg_Act	:ComSerialConfig:=(Baudrate:=0,Parity:=-1,RTS:=-1);(* internal used config struct - invalid initial values to ensure copying of input struct *)
	AdsSerialCfg1	:ComADSSerialConfig_1;		(* config struct which is transfered to Ads server *)
	pAdsSerialCfg	:XWORD;
	cbAdsSerialCfg	:UDINT;
	SrvName			:STRING(19);
	SrvVer			:UDINT;
	SrvVer_Act		:UDINT;

	State			:INT		:= STATE_WAIT;
	StateLast		:INT		:= STATE_WAIT;

	(* Only set one of the following triggers  on 'TRUE' at the same time! Wait until 'bBusy' is 'FALSE' again. *)
	ExeOpenPort		:BOOL		:= FALSE;		(* Set this value to 'TRUE' to perform the "Open serial port"-operation *)
	ExeCheckPort	:BOOL		:= FALSE;		(* Set this value to 'TRUE' to perform the "Check if  port is opened"-operation *)
	ExeWriteData	:BOOL		:= FALSE;		(* Set this value to 'TRUE' to perform the "Write data to port"-operation *)
	ExeCheckForData	:BOOL		:= FALSE;		(* Set this value to 'TRUE' to perform the "Check if serial port has buffered data"-operation *)
	ExeReadData		:BOOL		:= FALSE;		(* Set this value to 'TRUE' to perform the "Read out serial port"-operation *)
	ExeClosePort	:BOOL		:= FALSE;		(* Set this value to 'TRUE' to perform the "Close serial port"-operation *)
	ExeCheckVersion	:BOOL		:= FALSE;

	pWriteData		:XWORD;						(* Pointer to Data to write on serial port *)
	cbWriteData		:UDINT;						(* Length of data to write on serial port *)
	pReadData		:XWORD;						(* Pointer to Buffer for the read-data of serial port *)
	cbReadData		:UDINT;						(* Length of buffer for the read-data of serial port *)
	cbDataWaiting	:UDINT		:= 0;			(* Indicates the number of bytes waiting in the buffer of serial port *)

	AdsBusy			:BOOL		:= FALSE;		(* This output remains TRUE until the block has executed a command *)
	AdsError		:BOOL       := FALSE;       (* 'TRUE' if an error occured *)
	AdsErrorID		:UDINT      := 0;           (* Displays the error code; 0 = no error *)
	AdsCount		:UDINT		:= 0;			(* Displays the number of bytes read out by the ADSREADEX-functions *)

	(* TcSystem.lib has to be added for the following functions *)
	AdsWR_OpenPort		:ADSWRITE;
	AdsWR_WriteData		:ADSWRITE;
	AdsWR_ClosePort		:ADSWRITE;
	AdsRD_CheckPort		:ADSREADEX;
	AdsRD_CheckForData	:ADSREADEX;
	AdsRD_ReadData		:ADSREADEX;
	AdsRD_CheckVersion	:ADSRDDEVINFO;

	(* internal buffers (FiFo) *)
	RxBufferInt			:ARRAY[0..BUFFERSIZE_M1] OF BYTE;
	cbRxBufferInt		:UDINT;					(* number of bytes of valid data which need to be transfered *)
	TxBufferInt			:ARRAY[0..BUFFERSIZE_M1] OF BYTE;
	cbTxBufferInt		:UDINT;					(* number of bytes of valid data which need to be transfered *)

	cbTxCopyData		:UINT;
	cbRxCopyData		:UINT;

	iTemp				:UINT;

	timerDelayAfterErr	:TON:=(PT:=T#100ms);
	BlockedAfterErr		:BOOL;

	ErrInit				:UDINT;	(* for usage of error code constants to avoid warnings of unsued variables *)
END_VAR
{library private}
VAR CONSTANT
	BUFFERSIZE_M1		:UDINT	:= 1999;		(* -> internal buffer size 2000 bytes; buffer of server has to be bigger than buffer in Plc! *)
(*	BUFFERSIZESERVER	:UDINT	:= 10000;	*)	(* internal buffer size of ads server: 10000 bytes *)

	SERVERPORT			:UINT	:= 22122;		(* Port of the 'AdsSerialCommServer' *)
	MINSRVVER			:UDINT	:= 16#0201000D;	(* v2.1.13; minimum required server version; previous versions were beta and are not supported *)

	STATE_WAIT			:INT	:= 0;
	STATE_OPENPORT		:INT	:= ASC_CMD_OPENPORT;
	STATE_CHECKPORT		:INT	:= ASC_CMD_CHECKPORT;
	STATE_CLOSEPORT		:INT	:= ASC_CMD_CLOSEPORT;
	STATE_CHECKFORDATA	:INT	:= ASC_CMD_CHECKFORDATA;
	STATE_READDATA		:INT	:= ASC_CMD_READDATA;
	STATE_WRITEDATA		:INT	:= ASC_CMD_WRITEDATA;
	STATE_INIT			:INT	:= 7;

	WIN32_ERR_PREFIX	:UDINT	:=16#3D090000;
END_VAR

(* update ComBuffer - TxBuffer to arrTxBufferInt *)
IF NOT TxBuffer.blocked THEN
	Txbuffer.blocked  := TRUE;	(* block other PLC Tasks *)
	Txbuffer.FreeByte := SIZEOF(Txbuffer.Buffer) - Txbuffer.Count;
	cbTxCopyData      := MIN(TxBuffer.Count, SIZEOF(TxBufferInt) - UDINT_TO_UINT(cbTxBufferInt));
	IF cbTxCopyData > 0 THEN
		IF SIZEOF(TxBuffer.Buffer) < TxBuffer.RdIdx + cbTxCopyData THEN
			(* Tx Overrun *)
			iTemp := SIZEOF(TxBuffer.Buffer) - TxBuffer.RdIdx;
			MEMCPY(ADR(TxBufferInt)+cbTxBufferInt, ADR(TxBuffer.Buffer[TxBuffer.RdIdx]), iTemp );
			MEMCPY(ADR(TxBufferInt)+cbTxBufferInt+iTemp, ADR(TxBuffer.Buffer[0]), cbTxCopyData-iTemp);
			TxBuffer.RdIdx := TxBuffer.RdIdx + cbTxCopyData - SIZEOF(TxBuffer.Buffer);
		ELSE
			(* no Tx Overrun *)
			MEMCPY(ADR(TxBufferInt)+cbTxBufferInt, ADR(TxBuffer.Buffer[TxBuffer.RdIdx]), cbTxCopyData);
			TxBuffer.RdIdx := TxBuffer.RdIdx + cbTxCopyData;
			IF TxBuffer.RdIdx >= 301 THEN
				TxBuffer.RdIdx := 0;
			END_IF
		END_IF
		cbTxBufferInt     := cbTxBufferInt     + cbTxCopyData;
		TxBuffer.Count    := TxBuffer.Count    - cbTxCopyData;
		TxBuffer.FreeByte := TxBuffer.FreeByte + cbTxCopyData;
	END_IF
	Txbuffer.blocked := FALSE;	(* unblock other PLC Tasks *)
END_IF

Error   := FALSE;
ErrorId := 0;

(* state machine *)
CASE State OF
STATE_INIT:	(* first state - check version of TcAdsSerialCommServer *)
	IF NOT Busy THEN
		ExeCheckVersion := TRUE;
		AdsRD_CheckVersion(RDINFO := FALSE);
		Timeout_Act := Timeout;

		NetId_Act := NetId;			(* allocate new input value *)
	END_IF
	StateLast := State;
	(* Check the TcAdsSerialCommServer version to choose the right config structure in a later state *)
	AdsRD_CheckVersion(NETID:= NetId_Act,
					PORT	:= SERVERPORT,
					RDINFO	:= ExeCheckVersion,
					TMOUT	:= Timeout_Act,
					BUSY	=> AdsBusy,
					ERR		=> AdsError,
					ERRID	=> AdsErrorID,
					DEVNAME	=> SrvName,
					DEVVER	=>
	);
	IF NOT AdsBusy THEN
		Error   := AdsError;
		ErrorID := AdsErrorID;

		MEMCPY(ADR(SrvVer)+3, ADR(AdsRD_CheckVersion.DEVVER)  , 1);	(* copy version 1byte *)
		MEMCPY(ADR(SrvVer)+2, ADR(AdsRD_CheckVersion.DEVVER)+1, 1);	(* copy revision 1byte *)
		MEMCPY(ADR(SrvVer)  , ADR(AdsRD_CheckVersion.DEVVER)+2, 2);	(* copy build 2byte *)

		IF Error THEN
			NetId_Act := 'invalid';		(* invalid NetId to force INIT state again *)
		ELSIF SrvVer < MINSRVVER THEN		(* required minimum version of the ads server *)
			Error   := TRUE;
			ErrorID := COMERRORADS_SERVER_INCOMPATIBLE;
			NetId_Act := 'invalid';		(* invalid NetId to force INIT state again *)
		END_IF
		State := STATE_WAIT;
	END_IF
STATE_WAIT:	(* standard state if no new data is available on both sides *)
	StateLast := State;
	(* no ADS comm. *)
	IF NOT Busy AND NOT BlockedAfterErr THEN
		IF PortOpened THEN
			IF MEMCMP(ADR(SerialCfg),ADR(SerialCfg_Act),SIZEOF(SerialCfg)) <> 0	(* SerialCfg input changed *)
				OR NetId <> NetId_Act													(* NetId input changed *)
				OR NOT Connect THEN													(* disconnection requested *)
				State := STATE_CLOSEPORT;		(* close port and open again with new parameters *)
				cbTxBufferInt := 0;			(* reset internal buffer *)
			ELSE
				IF cbTxBufferInt > 0 THEN
					State := STATE_WRITEDATA;
				ELSE
					State := STATE_CHECKFORDATA;
				END_IF
			END_IF
		ELSE
			IF Connect THEN
				IF NetId <> NetId_Act	THEN	(* NetId input changed *)
					State := STATE_INIT;
				ELSE
					State := STATE_OPENPORT;
				END_IF
			END_IF
		END_IF
	END_IF
STATE_CHECKFORDATA:
	IF State <> StateLast THEN
		ExeCheckForData	:= TRUE;
		AdsRD_CheckForData(READ	:= 	FALSE);
		Timeout_Act := Timeout;
	END_IF
	StateLast := State;
	(* Check if serial port has buffered data *)
	AdsRD_CheckForData(NETID	:=	NetId_Act,
					PORT		:=	SERVERPORT,
					IDXGRP		:=	SerialCfg_Act.ComPort,
					IDXOFFS		:=	ASC_CMD_CHECKFORDATA,
					LEN			:=	SIZEOF(cbDataWaiting),
					DESTADDR	:=	ADR(cbDataWaiting),
					READ		:=	ExeCheckForData,
					TMOUT		:=	Timeout_Act,
					BUSY		=>	AdsBusy,
					ERR			=>	AdsError,
					ERRID		=>	AdsErrorID,
					COUNT_R		=>	AdsCount
	);
	IF NOT AdsBusy THEN
		Error   := AdsError;
		ErrorID := AdsErrorID;
		IF Error AND ErrorID = COMERRORADS_WR_FAILURE THEN
			StateLast := STATE_WAIT;	(* keep current state to repeat ads command *)
		ELSIF Error AND (ErrorID = COMERRORADS_PORT_NOT_CONNECTED OR ErrorID = COMERRORADS_RD_FAILURE) THEN (* port not yet opened -> open again *)
			PortOpened := FALSE;
			State      := STATE_OPENPORT;
		ELSIF Error AND ErrorID = COMERRORADS_RD_BUFFER_OVERRUN THEN
			IF cbDataWaiting = 0 THEN					(* ads command did not return data because of error *)
				cbDataWaiting:= SIZEOF(RxBufferInt);	(* buffer of server has to be bigger than buffer in Plc! *)
			END_IF
			State := STATE_READDATA;
		ELSIF NOT Error AND cbDataWaiting > 0 THEN
			State := STATE_READDATA;
		ELSE
			State := STATE_WAIT;
		END_IF
	END_IF
STATE_READDATA:
	IF State <> StateLast THEN
		ExeReadData := TRUE;
		AdsRD_ReadData(READ := FALSE);
		Timeout_Act := Timeout;
		(* allocate pointer *)
		pReadData  := ADR(RxBufferInt)+cbRxBufferInt;
		cbReadData := MIN(SIZEOF(RxBufferInt)-cbRxBufferInt, cbDataWaiting);	(* otherwise many zeros are transmitted - perhaps a failure of the server? *)
	END_IF
	StateLast := State;
	(* Read out serial port *)
	AdsRD_ReadData(	NETID		:=	NetId_Act,
					PORT		:=	SERVERPORT,
					IDXGRP		:=	SerialCfg_Act.ComPort,
					IDXOFFS		:=	ASC_CMD_READDATA,
					LEN			:=	cbReadData,
					DESTADDR	:=	pReadData,
					READ		:=	ExeReadData,
					TMOUT		:=	Timeout_Act,
					BUSY		=>	AdsBusy,
					ERR			=>	AdsError,
					ERRID		=>	AdsErrorID,
					COUNT_R		=>	AdsCount
	);
	IF NOT AdsBusy THEN
		Error   := AdsError;
		ErrorID := AdsErrorID;
		IF Error AND ErrorID = COMERRORADS_WR_FAILURE THEN
			StateLast := STATE_WAIT;	(* keep current state to repeat ads command *)
		ELSIF Error AND (ErrorID = COMERRORADS_PORT_NOT_CONNECTED OR ErrorID = COMERRORADS_RD_FAILURE) THEN (* port not yet opened -> open again *)
			PortOpened := FALSE;
			State      := STATE_OPENPORT;
		ELSE
			State := STATE_WAIT;
			IF NOT Error THEN
				(* allocate new buffer parameter *)
				IF (ADR(RxBufferInt)+cbRxBufferInt) <> pReadData THEN	(* internal buffer changed during ADS communication, new data copy necessary *)
					MEMCPY(ADR(RxBufferInt)+cbRxBufferInt, pReadData, AdsCount);
				END_IF
				cbRxBufferInt := cbRxBufferInt + AdsCount;
			END_IF
		END_IF
	END_IF
STATE_WRITEDATA:
	IF State <> StateLast THEN
		ExeWriteData := TRUE;
		AdsWR_WriteData(WRITE := FALSE);
		Timeout_Act := Timeout;
		(* allocate pointer *)
		pWriteData  := ADR(TxBufferInt);
		cbWriteData := MIN(cbTxBufferInt, SIZEOF(TxBufferInt));
	END_IF
	StateLast := State;
	(* "Write data to port *)
	AdsWR_WriteData(NETID		:=	NetId_Act,
					PORT		:=	SERVERPORT,
					IDXGRP		:=	SerialCfg_Act.ComPort,
					IDXOFFS		:=	ASC_CMD_WRITEDATA,
					LEN			:=	cbWriteData,
					SRCADDR		:=	pWriteData,
					WRITE		:= 	ExeWriteData,
					TMOUT		:=	Timeout_Act,
					BUSY		=>	AdsBusy,
					ERR			=>	AdsError,
					ERRID		=>	AdsErrorID
	);
	IF NOT AdsBusy THEN
		Error   := AdsError;
		ErrorID := AdsErrorID;
		IF Error AND ErrorID = COMERRORADS_WR_FAILURE THEN
			StateLast := STATE_WAIT;	(* keep current state to repeat ads command *)
		ELSIF Error AND (ErrorID = COMERRORADS_PORT_NOT_CONNECTED OR ErrorID = COMERRORADS_RD_FAILURE) THEN (* port not yet opened -> open again *)
			PortOpened := FALSE;
			State      := STATE_OPENPORT;
		ELSIF Error THEN
			State := STATE_WAIT;
		ELSE (* NOT bError *)
			State := STATE_CHECKFORDATA;
			(* release space of internal buffer (shift the rest to the front of the array) *)
			cbTxBufferInt := cbTxBufferInt - cbWriteData;
			IF cbTxBufferInt <> 0 THEN
				MEMCPY(ADR(TxBufferInt), ADR(TxBufferInt)+cbWriteData, cbTxBufferInt);
			END_IF
		END_IF
	END_IF
STATE_CHECKPORT:
	IF State <> StateLast THEN
		ExeCheckPort := TRUE;
		AdsRD_CheckPort(READ	:= 	FALSE);
		Timeout_Act := Timeout;
	END_IF
	StateLast := State;
	(* Check if serial port is already opened by the TcAdsSerialCommServer itselfs *)
	AdsRD_CheckPort(NETID		:=	NetId_Act,
					PORT		:=	SERVERPORT,
					IDXGRP		:=	SerialCfg_Act.ComPort,
					IDXOFFS		:=	ASC_CMD_CHECKPORT,
					LEN			:=	SIZEOF(PortOpened),
					DESTADDR	:=	ADR(PortOpened),
					READ		:=	ExeCheckPort,
					TMOUT		:=	Timeout_Act,
					BUSY		=>	AdsBusy,
					ERR			=>	AdsError,
					ERRID		=>	AdsErrorID,
					COUNT_R		=>	AdsCount
	);
	IF NOT AdsBusy THEN
		Error   := AdsError;
		ErrorID := AdsErrorID;
		IF Error AND ErrorID = COMERRORADS_WR_FAILURE THEN
			StateLast := STATE_WAIT;	(* keep current state to repeat ads command *)
		ELSIF Error AND ErrorID = COMERRORADS_RD_FAILURE THEN
			PortOpened := FALSE;
			State := STATE_WAIT;
		ELSE
			State := STATE_WAIT;
		END_IF
	END_IF
STATE_OPENPORT:
	IF State <> StateLast THEN
		ExeOpenPort := TRUE;
		AdsWR_OpenPort(WRITE := FALSE);
		Timeout_Act := Timeout;

		IF MEMCMP(ADR(SerialCfg), ADR(SerialCfg_Act), SIZEOF(SerialCfg)) <> 0 THEN	(* SerialCfg input changed *)
			MEMCPY(ADR(SerialCfg_Act), ADR(SerialCfg), SIZEOF(SerialCfg));			(* allocate new input configuration values *)
		END_IF

		SrvVer_Act := SrvVer;														(* allocate (new) received server version *)
		(* convert parameters input to internal AdsSerialCfg Server struct *)
		IF SrvVer >= MINSRVVER AND SrvVer < 16#FFFFFFFF THEN
			(* stAdsSerialCfg1.nStructVer;		- 1.structure version - initialized in structure declaration *)
			AdsSerialCfg1.TL		:= BYTE_TO_UINT(SerialCfg_Act.TraceLevel);
			AdsSerialCfg1.Baudrate	:= SerialCfg_Act.Baudrate;
			IF SerialCfg_Act.Parity = PARITY_EVEN THEN	(* Even and odd of parity in dcb API is switched *)
				AdsSerialCfg1.Parity := PARITY_ODD;
			ELSIF SerialCfg_Act.Parity = PARITY_ODD THEN
				AdsSerialCfg1.Parity := PARITY_EVEN;
			ELSE
				AdsSerialCfg1.Parity := SerialCfg_Act.Parity;
			END_IF
			AdsSerialCfg1.DataBits	:= SerialCfg_Act.DataBits;
			IF SerialCfg_Act.StopBits = STOPBITS_ONE THEN
				AdsSerialCfg1.StopBits := 0;
			ELSIF SerialCfg_Act.StopBits = STOPBITS_ONE5 THEN
				AdsSerialCfg1.StopBits := 1;
			ELSE
				AdsSerialCfg1.StopBits := SerialCfg_Act.StopBits;
			END_IF
			AdsSerialCfg1.DTR		:= SerialCfg_Act.DTR;
			AdsSerialCfg1.RTS		:= SerialCfg_Act.RTS;
			AdsSerialCfg1.CTS_Out	:= SerialCfg_Act.CTS;
			AdsSerialCfg1.DSR_Out	:= SerialCfg_Act.DSR;
			AdsSerialCfg1.DSR_Sens	:= SerialCfg_Act.DSR;
			pAdsSerialCfg			:= ADR(AdsSerialCfg1);
			cbAdsSerialCfg			:= SIZEOF(AdsSerialCfg1);
		END_IF
	END_IF
	StateLast := State;
	(* Open serial port *)
	AdsWR_OpenPort(	NETID		:=	NetId_Act,
					PORT		:=	SERVERPORT,
					IDXGRP		:=	SerialCfg_Act.ComPort,
					IDXOFFS		:=	ASC_CMD_OPENPORT,
					LEN			:=	cbAdsSerialCfg,
					SRCADDR		:=	pAdsSerialCfg,
					WRITE		:= 	ExeOpenPort,
					TMOUT		:=	Timeout_Act,
					BUSY		=>	AdsBusy,
					ERR			=>	AdsError,
					ERRID		=>	AdsErrorID
	);
	IF NOT AdsBusy THEN
		Error   := AdsError;
		ErrorID := AdsErrorID;
		IF Error AND ErrorID = COMERRORADS_WR_FAILURE THEN
			StateLast := STATE_WAIT;	(* keep current state to repeat ads command *)
		ELSIF Error AND ErrorID = COMERRORADS_PORT_CONNECTED THEN
			State := STATE_CLOSEPORT;	(* port already open -> close it and open again *)
		ELSE
			State := STATE_CHECKPORT;
		END_IF
	END_IF
STATE_CLOSEPORT:
	IF State <> StateLast THEN
		ExeClosePort := TRUE;
		AdsWR_ClosePort(WRITE := FALSE);
		Timeout_Act := Timeout;
	END_IF
	StateLast := State;
	(*Close serial port *)
	AdsWR_ClosePort(NETID		:=	NetId_Act,
					PORT		:=	SERVERPORT,
					IDXGRP		:=	SerialCfg_Act.ComPort,
					IDXOFFS		:=	ASC_CMD_CLOSEPORT,
					LEN			:=	cbAdsSerialCfg,
					SRCADDR		:=	pAdsSerialCfg,
					WRITE		:= 	ExeClosePort,
					TMOUT		:=	Timeout_Act,
					BUSY		=>	AdsBusy,
					ERR			=>	AdsError,
					ERRID		=>	AdsErrorID
	);
	IF NOT AdsBusy THEN
		Error   := AdsError;
		ErrorID := AdsErrorID;
		IF Error AND ErrorID = COMERRORADS_WR_FAILURE THEN
			StateLast := STATE_WAIT;	(* keep current state to repeat ads command *)
		ELSE
			PortOpened := FALSE;		(* also if the port is not closed successfully for example *)
			State := STATE_CHECKPORT;
		END_IF
	END_IF
END_CASE

Busy := AdsBusy;

(* Reset all triggers *)
ExeOpenPort     :=FALSE;
ExeCheckPort    :=FALSE;
ExeWriteData    :=FALSE;
ExeCheckForData :=FALSE;
ExeReadData     :=FALSE;
ExeClosePort    :=FALSE;
ExeCheckVersion :=FALSE;

(* update ComBuffer - arrRxBufferInt to RxBuffer *)
IF NOT RxBuffer.blocked THEN
	Rxbuffer.blocked  := TRUE;	(* block other PLC Tasks *)
	Rxbuffer.FreeByte := SIZEOF(Rxbuffer.Buffer) - Rxbuffer.Count;
	cbRxCopyData      := MIN(RxBuffer.FreeByte, UDINT_TO_UINT(cbRxBufferInt));
	IF cbRxCopyData > 0 THEN
		IF SIZEOF(RxBuffer.Buffer) < RxBuffer.WrIdx + cbRxCopyData THEN
			(* Rx Overrun *)
			iTemp := SIZEOF(RxBuffer.Buffer) - RxBuffer.WrIdx;
			MEMCPY(ADR(RxBuffer.Buffer[RxBuffer.WrIdx]), ADR(RxBufferInt), iTemp );
			MEMCPY(ADR(RxBuffer.Buffer[0]), ADR(RxBufferInt)+iTemp, cbRxCopyData-iTemp);
			RxBuffer.WrIdx := RxBuffer.WrIdx + cbRxCopyData - SIZEOF(RxBuffer.Buffer);
		ELSE
			(* no Rx Overrun *)
			MEMCPY(ADR(RxBuffer.Buffer[RxBuffer.WrIdx]), ADR(RxBufferInt), cbRxCopyData);
			RxBuffer.WrIdx := RxBuffer.WrIdx + cbRxCopyData;
			IF RxBuffer.WrIdx >= 301 THEN
				RxBuffer.WrIdx := 0;
			END_IF
		END_IF
		cbRxBufferInt     := cbRxBufferInt     - cbRxCopyData;
		RxBuffer.Count    := RxBuffer.Count    + cbRxCopyData;
		RxBuffer.FreeByte := RxBuffer.FreeByte - cbRxCopyData;
		(* release space of internal buffer (shift the rest to the front of the array) *)
		IF cbRxBufferInt <> 0 THEN
			MEMCPY(ADR(RxBufferInt), ADR(RxBufferInt)+cbRxCopyData, cbRxBufferInt);
		END_IF
	END_IF
	Rxbuffer.blocked := FALSE;	(* unblock other PLC Tasks *)
END_IF

TxBufCount := cbTxBufferInt;
RxBufCount := cbRxBufferInt;

(* stop ads communication for 100ms after win32 error *)
timerDelayAfterErr();
IF ErrorID >= WIN32_ERR_PREFIX AND NOT timerDelayAfterErr.Q THEN
	timerDelayAfterErr.IN := TRUE;
	BlockedAfterErr := TRUE;
END_IF
timerDelayAfterErr();
IF timerDelayAfterErr.Q THEN
	timerDelayAfterErr.IN := FALSE;
	BlockedAfterErr := FALSE; (* release block after delay *)
END_IF

IF TRUE = FALSE THEN
	(* usage of error code constants to avoid warnings of unsued variables *)
	ErrInit := COMERRORADS_INVALID_COMPORT;
	ErrInit := COMERRORADS_INVALID_CMD;
	ErrInit := COMERRORADS_INVALID_DATAPOINTER;
	ErrInit := COMERRORADS_INVALID_CFGSTLEN;
	ErrInit := COMERRORADS_INVALID_CFGSTVER;
	ErrInit := COMERRORADS_INVALID_TL;
	ErrInit := COMERRORADS_INVALID_BAUDRATE;
	ErrInit := COMERRORADS_INVALID_PARITY;
	ErrInit := COMERRORADS_INVALID_DATABITS;
	ErrInit := COMERRORADS_INVALID_STOPBITS;
	ErrInit := COMERRORADS_INVALID_DTR_CTRL;
	ErrInit := COMERRORADS_INVALID_RTS_CTRL;
	ErrInit := COMERRORADS_INVALID_CTS_OUTCTRL;
	ErrInit := COMERRORADS_INVALID_DSR_OUTCTRL;
	ErrInit := COMERRORADS_INVALID_DSR_SENS;
	ErrInit := COMERRORADS_NOT_INIT;
	ErrInit := COMERRORADS_RD_BUFFER_OVERRUN;
	ErrInit := COMERRORADS_PORT_CONNECTED;
	ErrInit := COMERRORADS_PORT_NOT_CONNECTED;
	ErrInit := COMERRORADS_RD_THREAD_TIMEOUT;
	ErrInit := COMERRORADS_WR_THREAD_TIMEOUT;
	ErrInit := COMERRORADS_RD_FAILURE;
	ErrInit := COMERRORADS_WR_FAILURE;
	ErrInit := COMERRORADS_SERVER_INCOMPATIBLE;
END_IF

END_FUNCTION_BLOCK

// POUs/COMlibV2/Background Communication/SerialLineControlM8000
(* =============================================================
 *	Modul:	Serial line interface controller for background communication
 *			supports M8000 LightBus modules
 *			communication between a serial line hardware device and 
 *			PLC communication buffers (RxBuffer, TxBuffer)
 *
 *	Date: 	01.09.2009
 * ============================================================= *)
FUNCTION_BLOCK SerialLineControlM8000
VAR_INPUT
	Channel : INT;
	pComIn : 	POINTER TO ARRAY[0..65] OF BYTE; (* must meet the maximum size of a hardware related data structure *)
	pComOut :	POINTER TO ARRAY[0..65] OF BYTE; (* must meet the maximum size of a hardware related data structure *)
	SizeComIn :	UINT;
END_VAR
VAR_OUTPUT
	Error : BOOL;
	ErrorID : ComError_t;
END_VAR
VAR_IN_OUT
	TxBuffer 	:	COMbuffer;
	RxBuffer :	COMbuffer;
END_VAR
VAR
	ComPortDebugBuffer:ComDebugBuffer;
	InvalidDataExchangeMode: UINT;
	CommandMode: UINT;
	pCTRL: POINTER TO BYTE;
	pSTATUS: POINTER TO BYTE;
	TransmitBufferFullBit: BYTE;
	TransmitDataValidBit: BYTE;
	ReceiveDataValidBit: BYTE;
(*	noTAcounter: BYTE;*)
	initialized: BOOL;
(*	i: INT;*)
	TransmitBufferSentBit: BYTE;
END_VAR

IF pComIn=0 OR pComOut=0 OR SizeComIn=0 THEN
	Error := TRUE;
	ErrorID := COMERROR_INVALIDPOINTER;
	RETURN;
ELSIF SizeComIn<>4 THEN
	Error := TRUE;
	ErrorID := COMERROR_INVALIDPROCESSDATASIZE;
	RETURN;
ELSIF Channel < 1 OR Channel > 3 THEN
	Error := TRUE;
	ErrorID := COMERROR_INVALIDCHANNELNUMBER;
	RETURN;
ELSE
	Error := FALSE;
	ErrorID := 0;
END_IF

(* pointer to I/O data structures *)
pCTRL := pComOut+3;
pSTATUS := pComIn+3;

InvalidDataExchangeMode := 	(pCTRL^ 	AND 2#11000000) OR	(* command mode *)
							(pSTATUS^	AND 2#01000000);		(* command mode *)

CommandMode 		:= 		(pCTRL^ 	AND 2#10000000);

TransmitBufferSentBit 	:= 		2#10000000;	(* *)

CASE Channel OF
	1 :	ReceiveDataValidBit	:= 	2#00000001;
		TransmitDataValidBit	:= 	2#00000001;
		TransmitBufferFullBit	:= 	2#00001000;
	2 :	ReceiveDataValidBit	:= 	2#00000010;
		TransmitDataValidBit	:= 	2#00000010;
		TransmitBufferFullBit	:= 	2#00010000;
	3 :	ReceiveDataValidBit	:= 	2#00000100;
		TransmitDataValidBit	:= 	2#00000100;
		TransmitBufferFullBit	:= 	2#00100000;
END_CASE

initialized := TRUE;

IF initialized THEN
	IF  InvalidDataExchangeMode = 0 THEN (* don't talk to the terminal during reset or register access *)

		(* Read data from serial interface to RxBuffer *)
		IF NOT RXbuffer.blocked THEN (* check if the buffer is blocked by the standard PLC task *)
			RXbuffer.FreeByte := SIZEOF(RXbuffer.Buffer) - RXbuffer.Count;
			IF ((pSTATUS^ AND ReceiveDataValidBit) <> 0) AND RxBuffer.FreeByte >= 1THEN
				(* copy data byte from the I/O buffer *)
				RXbuffer.Buffer[RXbuffer.WrIdx] := pComIn^[Channel-1];
				RXbuffer.WrIdx := RXbuffer.WrIdx + 1;
				IF RXbuffer.WrIdx >= SIZEOF(RXbuffer.Buffer) THEN
					RXbuffer.WrIdx := 0;
				END_IF
				(* copy data byte the the debug buffer *)
				ComPortDebugBuffer.Buffer[ComPortDebugBuffer.Idx]:=BYTE_TO_INT(pComIn^[Channel-1]);
				ComPortDebugBuffer.Status[ComPortDebugBuffer.Idx]:=1;
				IF UINT_TO_INT(ComPortDebugBuffer.Idx) < BUFFERSIZE_DEBUGBUFFER THEN
					ComPortDebugBuffer.Idx := ComPortDebugBuffer.Idx + 1;
				ELSE
					ComPortDebugBuffer.Idx:=0;
				END_IF
				RXbuffer.Count := RXbuffer.Count + 1;
				RXbuffer.FreeByte := SIZEOF(RXbuffer.Buffer) - RXbuffer.Count;
			END_IF
		END_IF

		(* Write data TxBuffer to serial interface *)
		IF ((pSTATUS^ AND TransmitBufferSentBit) <> 0) THEN (* transmit buffer sent - if zero keep telegram unchanged and repeat it *)
			pCTRL^ := pCTRL^ AND NOT TransmitDataValidBit;	(* no data to send - default *)
			IF NOT TXbuffer.blocked AND ((pSTATUS^ AND TransmitBufferFullBit)=0) THEN
				IF TxBuffer.Count > 0 THEN (* check if the buffer is blocked by the standard PLC task *)
					(* copy data byte to the I/O buffer *)
					pComOut^[Channel-1] := TxBuffer.Buffer[TXbuffer.RdIdx];
					TXbuffer.RdIdx := TXbuffer.RdIdx + 1;
					IF TXbuffer.RdIdx >= SIZEOF(TXbuffer.Buffer) THEN
						TXbuffer.RdIdx := 0;
					END_IF
					(* copy data byte the the debug buffer *)
					ComPortDebugBuffer.Buffer[ComPortDebugBuffer.Idx]:=BYTE_TO_INT(pComOut^[Channel-1]);
					ComPortDebugBuffer.Status[ComPortDebugBuffer.Idx]:=2;
					IF UINT_TO_INT(ComPortDebugBuffer.Idx) < BUFFERSIZE_DEBUGBUFFER THEN
						ComPortDebugBuffer.Idx := ComPortDebugBuffer.Idx + 1;
					ELSE
						ComPortDebugBuffer.Idx:=0;
					END_IF
					TXbuffer.Count := TXbuffer.Count - 1;
					TXbuffer.FreeByte := SIZEOF(TXbuffer.Buffer) - TXbuffer.Count;
					pCTRL^ := pCTRL^ XOR TransmitDataValidBit; (* toggle transmit data valid bit *)
				END_IF
			END_IF
		END_IF
	END_IF
END_IF

END_FUNCTION_BLOCK

// POUs/COMlibV2/CO_Nfiguration/KL6configuration
FUNCTION_BLOCK KL6configuration
VAR_INPUT
	Execute		: BOOL;
	Mode 		: ComSerialLineMode_t;
	Baudrate		: UDINT;			(*	115200, 57600, 38400, 19200, 9600, 4800, 2400, 1200, 600, 300 *)
	NoDatabits	: BYTE;			(*	7 or 8 *)
	Parity		: ComParity_t;		(*	PARITY_NONE=0, PARITY_EVEN=1, PARITY_ODD=2 *)
	Stopbits		: BYTE;			(*	1 or 2 *)
	Handshake	: ComHandshake_t;	(*	HANDSHAKE_NONE=0, HANDSHAKE_RTSCTS=1, HANDSHAKE_XONXOFF=2 *)
	ContinousMode : BOOL;		(* don't start transmission before transmit buffer is filled *)
	pComIn		: POINTER TO ARRAY[0..65] OF BYTE;	(* for universal register communication *)
	pComOut	: POINTER TO ARRAY[0..65] OF BYTE;	(* for universal register communication *)
	SizeComIn	: UINT;
END_VAR
VAR_OUTPUT
	Done 		: BOOL;
	Busy		: BOOL;
	Error		: BOOL;
	ErrorId		: ComError_t;
END_VAR
VAR CONSTANT
	TIME_OUT_VALUE	: TIME  := T#100MS;
	RESETMASK_STANDARD		: WORD := 2#00000100;
	RESETMASK_ALTERNATIVE	: WORD := 2#00000100_00000000;
	REGISTERACCESSMASK		: BYTE := 2#10000000;	(* 2011-09-12 KSt *)
END_VAR
VAR
	state: INT;
	TriggerExecute: R_TRIG;
	R32 : WORD;
	R33 : WORD;
	R34 : WORD;
	CheckOK: BOOL;
	RegisterList : ARRAY[31..35] OF ComRegisterData_t;
	WriteRegisterList: KL6WriteRegisters;
	Timeout: TON;
	pCTRL: POINTER TO WORD;
	pSTATUS: POINTER TO WORD;
	ResetMask : WORD;
END_VAR

TriggerExecute(CLK:=Execute);
CASE state OF
	0 : (* init *)
		Busy := FALSE;
		IF NOT Execute THEN
			Done := FALSE;
		END_IF
		IF TriggerExecute.Q THEN
			IF pComIn=0 OR pComOut=0 THEN
				Error := TRUE;
				ErrorID := COMERROR_INVALIDPOINTER;
			ELSE
				Done := FALSE;
				Error := FALSE;
				ErrorID := 0;
				CheckOK  := FALSE;
				pCTRL := pComOut;
				pSTATUS := pComIn;
				ResetMask := RESETMASK_STANDARD;
				WriteRegisterList(Execute:=FALSE);
				Timeout(IN:=FALSE);
				Busy := TRUE;
				state := state + 1;
			END_IF
		END_IF

	1: (* check parameter *)

		CASE Baudrate OF
			300 :		R32 := 2#00000001;	(* 2011-08-24 KSt - added *)
			600 :		R32 := 2#00000010;	(* 2011-08-24 KSt - added *)
			1200 :	R32 := 2#00000011;
			2400 :	R32 := 2#00000100;
			4800 :	R32 := 2#00000101;
			9600 :	R32 := 2#00000110;
			19200 :	R32 := 2#00000111;
			38400 :	R32 := 2#00001000;
			57600 :	R32 := 2#00001001;
			115200 :	R32 := 2#00001010;
			ELSE
				ErrorID := COMERROR_INVALIDBAUDRATE;
		END_CASE

		(* check number of databits, stopbits and parity *)
		IF (NoDatabits <> 8) AND (NoDatabits <> 7) THEN
			ErrorID := COMERROR_INVALIDNUMDATABITS;
		ELSE
			CASE Parity OF
				PARITY_NONE :
					IF NoDatabits = 7 THEN
						ErrorId := COMERROR_INVALIDPARITY;
					ELSE
						R33 := 2#0000011;   (* 8 Bit no Parity *)
					END_IF
				PARITY_ODD:
					R33 := SEL(NoDatabits=8,
								2#0000010,		(* 7 Bit, odd Parity *)
								2#0000101 );	(* 8 Bit, odd Parity *)
				PARITY_EVEN:
					R33 := SEL(NoDatabits=8,
								2#0000001,		(* 7 Bit, even Parity *)
								2#0000100 );	(* 8 Bit, even Parity *)
				ELSE
					ErrorId := COMERROR_INVALIDPARITY;
			END_CASE
		END_IF
		CASE Stopbits OF
			1 : R33 := R33 OR 2#00000000;
			2 : R33 := R33 OR 2#00001000;
			ELSE
				ErrorID := COMERROR_INVALIDNUMSTOPBITS;
		END_CASE

		CASE Handshake OF
			HANDSHAKE_NONE :				R34 := 2#00000000;
			HANDSHAKE_RTSCTS :			R34 := 2#00000001;
			HANDSHAKE_XONXOFF :			R34 := 2#00011000;
			RS485_HALFDUPLEX_XONXOFF :	R34 := 2#00011001; (* 15.11.2000 KSt *)
			RS485_HALFDUPLEX :			R34 := 2#00000001; (* same as RTS/CTS *)
			RS485_FULLDUPLEX :				R34 := 2#00000000; (* same as NONE *)
			RS485_FULLDUPLEX_XONXOFF :	R34 := 2#00011000; (* same as XON/XOFF *)
			ELSE
				ErrorId := COMERROR_INVALIDHANDSHAKE;
		END_CASE
		IF ContinousMode THEN
			R34 := R34 OR 2#01000000; (* continous mode *)
		END_IF
		IF SizeComIn = 5 THEN
			R34 := R34 OR 2#00000010; (* alternative mode *)
			ResetMask := RESETMASK_ALTERNATIVE;
		ELSIF SizeComIn >= 8 THEN
			(* KL6 long data size (22 byte) *)
			R34 := R34 OR 2#00000001_10000000; (* extend process data interface - optimized transfer rate *)
		END_IF

		(*******    EXIT ON ERROR CONDITIONif any error in the input then return to caller with the error code   ******)
		IF   ErrorId <> 0  THEN
			Error := TRUE;
			state := 0;
		ELSE
			RegisterList[31].Register := 31;
			RegisterList[31].Value := 16#1235;
			RegisterList[32].Register := 32;
			RegisterList[32].Value := R32;
			RegisterList[33].Register := 33;
			RegisterList[33].Value := R33;
			RegisterList[34].Register := 34;
			RegisterList[34].Value := R34;
			RegisterList[35].Register := 31;
			RegisterList[35].Value := 0;
			CheckOK  := TRUE;
			state := state + 1;
		END_IF

	2:	(* reset terminal *)
		pCTRL^ := ResetMask;
		Timeout(IN:=TRUE , PT:=TIME_OUT_VALUE );
		IF  ( pSTATUS^ AND ResetMask) <> 0 THEN
			pCTRL^ := pCTRL^ AND NOT RESETMASK;	(* 2011-08-24 KSt - added *)
			Timeout(IN:=FALSE);
  			state := state + 1;
		ELSIF Timeout.Q THEN
			pCTRL^ := pCTRL^ AND NOT RESETMASK;	(* 2011-08-24 KSt - added *)
			Error := TRUE;
			ErrorID := COMERROR_TIMEOUT;
			state := 0;
		END_IF

	3:	(* write R32 *)
		WriteRegisterList( 	Execute:=TRUE ,
							Mode:=Mode ,
							pComIn:=pComIn ,
							pComOut:=pComOut ,
							SizeComIn:=SizeComIn ,
							pRegisterList:=ADR(RegisterList) ,
							SizeRegisterList:=SIZEOF(RegisterList) );
		IF NOT WriteRegisterList.Busy THEN
			Error := WriteRegisterList.Error;
			ErrorID := WriteRegisterList.ErrorID;
			pCTRL^ := pCTRL^ AND NOT RESETMASK;
			state := state + 1;
		END_IF

	4:	(* reset terminal *)
		pCTRL^ := ResetMask;
		Timeout(IN:=TRUE , PT:=TIME_OUT_VALUE );
(*		IF  ( pSTATUS^ AND ResetMask) <> 0 THEN *)		(* 2011-09-12 KSt *)
		IF  ( pSTATUS^ AND (ResetMask OR REGISTERACCESSMASK) ) = ResetMask THEN		(* 2011-09-12 KSt *)
			(* 2011-09-12 KSt: check of REGISTERACCESSMASK avoids wrong feedback of Reset-Bit if register communication is still active *)
			Timeout(IN:=FALSE);
			pCTRL^ := pCTRL^ AND NOT RESETMASK;
  			state := state + 1;
		ELSIF Timeout.Q THEN
			pCTRL^ := pCTRL^ AND NOT RESETMASK;	(* 2011-08-24 KSt - added *)
			Error := TRUE;
			ErrorID := COMERROR_TIMEOUT;
			state := 0;
		END_IF

	5:	(* wait reset done *)
		Timeout(IN:=TRUE , PT:=TIME_OUT_VALUE );
		IF  ( pSTATUS^ AND ResetMask) = 0 THEN
			Timeout(IN:=FALSE);
			Done := NOT Error;
  			state := 0;
		ELSIF Timeout.Q THEN
			Error := TRUE;
			ErrorID := COMERROR_TIMEOUT;
			state := 0;
		END_IF
END_CASE

END_FUNCTION_BLOCK

// POUs/COMlibV2/CO_Nfiguration/KL6WriteRegisters
(*=============================================================
 *	Modul:	Write access to terminal registers
 *			supports multiple interface types like 
 *			KL6xxx 3 byte alternative mode
 *			KL6xxx 5 byte standard mode
 *			KL6xxx 22 byte standard mode with extended process data interface
 *			
 *	Date: 	21.12.2004
 *
 *=============================================================
 *)
FUNCTION_BLOCK KL6WriteRegisters
VAR_INPUT
	Execute	: BOOL;
	Mode : ComSerialLineMode_t;
	pComIn	: POINTER TO ARRAY[0..65] OF BYTE;	(* for universal register communication *)
	pComOut	: POINTER TO ARRAY[0..65] OF BYTE;	(* for universal register communication *)
	SizeComIn :	UINT;
	pRegisterList : POINTER TO ARRAY[0..63] OF ComRegisterData_t;
	SizeRegisterList : UINT;
END_VAR
VAR_OUTPUT
	Done 		: BOOL;
	Busy		: BOOL;
	Error		: BOOL;
	ErrorId		: ComError_t;
END_VAR
VAR CONSTANT
	TIME_OUT_VALUE		: TIME  := T#100MS;
	REGISTERNUMBERMASK : BYTE := 2#00111111;
	REGISTERWRITEMASK	: BYTE := 2#11000000;
END_VAR
VAR
	state: INT;
	TriggerExecute: R_TRIG;
	NumRegisters: UINT;
	n: UINT;
	Register: BYTE;
	Value: WORD;
	Timeout: TON;
	pCTRL: POINTER TO BYTE;
	pSTATUS: POINTER TO BYTE;
	SaveCTRL: BYTE;
END_VAR

TriggerExecute(CLK:=Execute);
CASE state OF
	0 : (* init *)
		Busy := FALSE;
		IF NOT Execute THEN
			Done := FALSE;
		END_IF
		IF TriggerExecute.Q THEN
			Error := FALSE;
			ErrorID := 0;
			NumRegisters := SizeRegisterList / SIZEOF(pRegisterList^[0]);
			IF pComIn=0 OR pComOut=0 THEN
				ErrorID := COMERROR_INVALIDPOINTER;
			ELSIF NumRegisters < 1 OR NumRegisters > 64 THEN
				ErrorID := COMERROR_INVALIDNUMREGISTERS;
			ELSE
				FOR n := 0 TO NumRegisters - 1 DO
					IF pRegisterList^[n].Register > 63 OR pRegisterList^[0].Register = 0 THEN
						ErrorID := COMERROR_INVALIDREGISTER;
						EXIT;
					END_IF
				END_FOR
				Error := ErrorID<>0;
				IF NOT Error THEN
					Done := FALSE;
					Error := FALSE;
					ErrorID := 0;
					Busy := TRUE;
					pCTRL := pComOut;
					pSTATUS := pComIn;
					SaveCTRL := pCTRL^;
					Timeout(IN:=FALSE);
					n := 0;
					state := state + 1;
				END_IF
			END_IF
		END_IF

	1: (* write registers *)
		Register := pRegisterList^[n].Register;
		IF Register=0 THEN
			pCTRL^ := SaveCTRL;
			Done := n>0;
			state := 0;
		ELSE
			Value := pRegisterList^[n].Value;
			pCTRL^ := REGISTERWRITEMASK + Register;
			pComOut^[1] := WORD_TO_BYTE( Value AND 2#11111111);
			pComOut^[2] := WORD_TO_BYTE( SHR(Value, 8) );
			state := state + 1;
		END_IF

	2:	(* Wait for positive confirmation *)
		Timeout(IN:=TRUE , PT:=TIME_OUT_VALUE );
		IF  ( pSTATUS^ AND REGISTERNUMBERMASK) = Register THEN
			Timeout(IN:=FALSE);
			n := n + 1;
			IF n >= NumRegisters THEN
				pCTRL^ := SaveCTRL;
				Done := TRUE;
				state := 0;
			ELSE
				state := 1;
			END_IF
		ELSIF Timeout.Q THEN
			pCTRL^ := SaveCTRL;
			Error := TRUE;
			ErrorID := COMERROR_TIMEOUT;
			state := 0;
		END_IF

END_CASE

END_FUNCTION_BLOCK

// POUs/COMlibV2/CO_Nfiguration/KL6ReadRegisters
(*=============================================================
 *	Modul:	Read access to terminal registers
 *			supports multiple interface types like 
 *			KL6xxx 3 byte alternative mode
 *			KL6xxx 5 byte standard mode
 *			KL6xxx 22 byte standard mode with extended process data interface
 *			
 *	Date: 	21.12.2004
 *
 *=============================================================
 *)
FUNCTION_BLOCK KL6ReadRegisters
VAR_INPUT
	Execute	: BOOL;
	FirstRegister : UINT;
	RegisterCount : UINT;
	Mode : ComSerialLineMode_t;
	pComIn	: POINTER TO ARRAY[0..65] OF BYTE;	(* for universal register communication *)
	pComOut	: POINTER TO ARRAY[0..65] OF BYTE;	(* for universal register communication *)
	SizeComIn :	UINT;
	pRegisterList : POINTER TO ARRAY[0..63] OF ComRegisterData_t;
	SizeRegisterList : UINT;
END_VAR
VAR_OUTPUT
	Done 		: BOOL;
	Busy		: BOOL;
	Error		: BOOL;
	ErrorId		: ComError_t;
END_VAR
VAR CONSTANT
	TIME_OUT_VALUE		: TIME  := T#100MS;
	REGISTERNUMBERMASK : BYTE := 2#00111111;
	REGISTERREADMASK	: BYTE := 2#10000000;
END_VAR
VAR
	state: INT;
	TriggerExecute: R_TRIG;
	NumRegisters: UINT;
	n: UINT;
	Register: BYTE;
	Value: WORD;
	Timeout: TON;
	pCTRL: POINTER TO BYTE;
	pSTATUS: POINTER TO BYTE;
(*	NumRegistersInList: INT;*)
	i: UINT;
	SaveCTRL: BYTE;
END_VAR

TriggerExecute(CLK:=Execute);
CASE state OF
	0 : (* init *)
		Busy := FALSE;
		IF NOT Execute THEN
			Done := FALSE;
		END_IF
		IF TriggerExecute.Q THEN
			Error := FALSE;
			ErrorID := 0;
			NumRegisters := SizeRegisterList / SIZEOF(pRegisterList^[0]);
			IF NumRegisters < RegisterCount THEN
				ErrorID := COMERROR_INVALIDNUMREGISTERS;
			ELSIF pComIn=0 OR pComOut=0 THEN
				ErrorID := COMERROR_INVALIDPOINTER;
			ELSIF NumRegisters < 1 OR NumRegisters > 64 OR RegisterCount < 1 OR RegisterCount > 64 THEN
				ErrorID := COMERROR_INVALIDNUMREGISTERS;
			ELSIF FirstRegister <> 16#FFFF AND (FirstRegister > 63 OR (FirstRegister + RegisterCount) > 64) THEN
				ErrorID := COMERROR_INVALIDREGISTER;
			ELSE
				IF FirstRegister <> 16#FFFF THEN (* initialize list with register numbers *)
					FOR i := 0 TO NumRegisters-1 DO
						pRegisterList^[i].Register := UINT_TO_BYTE( SEL( i >= RegisterCount, FirstRegister + i, 0));
					END_FOR
				ELSE (* use user defined register numbers in list *)
					FOR n := 0 TO NumRegisters - 1 DO
						IF pRegisterList^[n].Register > 63 THEN
							ErrorID := COMERROR_INVALIDREGISTER;
							EXIT;
						END_IF
					END_FOR
				END_IF
				Error := ErrorID <> 0;
				IF NOT Error THEN
					Done := FALSE;
					Error := FALSE;
					ErrorID := 0;
					Busy := TRUE;
					pCTRL := pComOut;
					pSTATUS := pComIn;
					SaveCTRL := pCTRL^;
					Timeout(IN:=FALSE);
					n := 0;
					state := state + 1;
				END_IF
			END_IF
		END_IF

	1:	(* read register and wait for positive confirmation *)
		Register := pRegisterList^[n].Register;
		pCTRL^ := REGISTERREADMASK + Register;
		Timeout(IN:=TRUE , PT:=TIME_OUT_VALUE );
		IF  ( pSTATUS^ AND REGISTERNUMBERMASK) = Register THEN
			Value := pComIn^[1] + 256*pComIn^[2];
			pRegisterList^[n].Value := Value;
			Timeout(IN:=FALSE);
			n := n + 1;
			IF n >= NumRegisters THEN
				pCTRL^ := SaveCTRL;
				Done := TRUE;
				state := 0;
			END_IF
		ELSIF Timeout.Q THEN
			pCTRL^ := SaveCTRL;
			Error := TRUE;
			ErrorID := COMERROR_TIMEOUT;
			state := 0;
		END_IF

END_CASE

END_FUNCTION_BLOCK

// POUs/COMlibV2/CO_Nfiguration/M8000configuration
FUNCTION_BLOCK M8000configuration
VAR_INPUT
	Execute		: BOOL;
	Channel		: INT;			(* 	1..3 *)
	Baudrate		: UDINT;			(*	115200, 57600, 38400, 19200, 9600, 4800, 2400, 1200 *)
	NoDatabits	: BYTE;			(*	7 or 8 *)
	Parity		: ComParity_t;		(*	PARITY_NONE=0, PARITY_EVEN=1, PARITY_ODD=2 *)
	Stopbits		: BYTE;			(*	1 or 2 *)
	Handshake	: ComHandshake_t;	(*	HANDSHAKE_NONE=0, HANDSHAKE_RTSCTS=1, HANDSHAKE_XONXOFF=2 *)
END_VAR
VAR_OUTPUT
	Done 		: BOOL;
	Busy		: BOOL;
	Error		: BOOL;
	ErrorId		: ComError_t;
END_VAR
VAR_IN_OUT
	ComIn	: M8000inData;	(* for universal register communication *)
	ComOut	: M8000outData;	(* for universal register communication *)
END_VAR
VAR
	state: INT;
	TriggerExecute: R_TRIG;
	TimerTimeout: TON;
END_VAR

TriggerExecute(CLK:=Execute);
TimerTimeout();

CASE state OF
	0 : 	(* wait for trigger *)
		Busy := FALSE;
		IF NOT Execute THEN
			Done := FALSE;
		END_IF
		IF TriggerExecute.Q THEN
			Busy := TRUE;
			Done := FALSE;
			Error := FALSE;
			ErrorID := 0;
			TimerTimeout(IN:=FALSE);
			TimerTimeout(IN:=TRUE, PT := T#1s);
			state := state +1;
		END_IF

	1 : 	(* wait for valid data exchange mode *)
		IF (ComOut.D[3] AND 2#11000000) = 0 THEN
			CASE Baudrate OF
				300:		ComOut.D[0] := 2#00110000;
				600:		ComOut.D[0] := 2#01000000;
				1200:	ComOut.D[0] := 2#01010000;
				2400:	ComOut.D[0] := 2#01100000;
				4800:	ComOut.D[0] := 2#10000000;
				9600:	ComOut.D[0] := 2#10010000;
				3600:	ComOut.D[0] := 2#10100000;
				19200:	ComOut.D[0] := 2#10110000;
				37400:	ComOut.D[0] := 2#11000000;
			ELSE
				ComOut.D[0] := 2#10110000; (* 19200 *)
				Error := TRUE;
				ErrorID := COMERROR_INVALIDBAUDRATE;
			END_CASE
			(* set number of stop bits *)
			CASE Stopbits OF
				1 : 	ComOut.D[0] := ComOut.D[0] OR 2#0111;
				2 : 	ComOut.D[0] := ComOut.D[0] OR 2#1111;
			ELSE
				ComOut.D[0] := ComOut.D[0] OR 2#0111;
				Error := TRUE;
				ErrorID := COMERROR_INVALIDNUMSTOPBITS;
			END_CASE
			(* set handshake *)
			CASE Handshake OF
				HANDSHAKE_RTSCTS :
					ComOut.D[1] := 2#000_00000;
				HANDSHAKE_XONXOFF :
					ComOut.D[1] := 2#001_00000;
(*				HANDSHAKE_NONE :
					ComOut.D[1] := 2#100_00000;*)	(* ??? Wert nicht bekannt, da in der Doku nicht beschrieben *)
			ELSE
				ComOut.D[1] := 2#000_00000;	(* HANDSHAKE_RTSCTS *)
				Error := TRUE;
				ErrorID := COMERROR_INVALIDHANDSHAKE;
			END_CASE
			(* set parity *)
			CASE Parity OF
				PARITY_NONE :	ComOut.D[1] := ComOut.D[1] OR 2#000_100_00;
				PARITY_EVEN :	ComOut.D[1] := ComOut.D[1] OR 2#000_000_00;
				PARITY_ODD :	ComOut.D[1] := ComOut.D[1] OR 2#000_001_00;
			ELSE
				ComOut.D[1] := ComOut.D[1] OR 2#000_100_00;
				Error := TRUE;
				ErrorID := COMERROR_INVALIDPARITY;
			END_CASE
			(* set number of data bits *)
			CASE NoDatabits OF
				7 :	ComOut.D[1] := ComOut.D[1] OR 2#10;
				8 :	ComOut.D[1] := ComOut.D[1] OR 2#11;
			ELSE
				ComOut.D[1] := ComOut.D[1] OR 2#11;
				Error := TRUE;
				ErrorID := COMERROR_INVALIDNUMDATABITS;
			END_CASE

			IF Error THEN
				state := 0;
			ELSE
				state := state +1;
				CASE Channel OF
					1 : 	ComOut.D[3] := ComOut.D[3] OR 2#01_000001;
					2 :	ComOut.D[3] := ComOut.D[3] OR 2#01_000010;
					3 :	ComOut.D[3] := ComOut.D[3] OR 2#01_000100;
				ELSE
					Error := TRUE;
					ErrorID := COMERROR_INVALIDCHANNELNUMBER;
					state := 0;
				END_CASE
			END_IF
		ELSIF TimerTimeout.Q THEN
			Error := TRUE;
			ErrorID := COMERROR_TIMEOUT;
			state := 0;
		END_IF

	2 : (* wait for initialization done *)
		IF ComIn.D[3].7 THEN
			ComOut.D[3] := 0;
			Done := TRUE;
			state := 0;
		ELSIF TimerTimeout.Q THEN
			Error := TRUE;
			ErrorID := COMERROR_TIMEOUT;
			state := 0;
		END_IF
END_CASE

IF state = 0 THEN
	Busy := FALSE;
END_IF

END_FUNCTION_BLOCK

// POUs/COMlibV2/Send + Receive/ReceiveData
FUNCTION_BLOCK ReceiveData
VAR_INPUT
	pPrefix : POINTER TO BYTE;
	LenPrefix : BYTE;
	pSuffix : POINTER TO BYTE;
	LenSuffix : BYTE;
	pReceiveData : POINTER TO BYTE;
	SizeReceiveData : UDINT;
	Timeout : TIME;
	Reset :BOOL;
END_VAR
VAR_OUTPUT
	DataReceived	: BOOL;
	busy 			: BOOL;
	Error			: ComError_t;
	RxTimeout 		: BOOL;
	LenReceiveData 	: UDINT;
END_VAR
VAR_IN_OUT
	RXbuffer 			: COMbuffer;
END_VAR
VAR
	state: UINT;
	c : BYTE;
	l : UINT;
	iTimeout : TIME;
	Receive : ReceiveByte;
	TimeoutTimer : TOF;
	ptrPrefix : POINTER TO BYTE;
	pData : POINTER TO BYTE;
	p1 : POINTER TO BYTE;
	p2 : POINTER TO BYTE;
	isEqual: BOOL;
	i: UINT;
	pw : XWORD;
END_VAR

IF Reset THEN
	state := 0;
	RETURN;
END_IF
IF pReceiveData = 0 THEN
	Error := COMERROR_INVALIDRXPOINTER;
	state := 0;
	RETURN;
END_IF
IF SizeReceiveData = 0 THEN
	Error := COMERROR_INVALIDRXLENGTH;
	state := 0;
	RETURN;
END_IF
IF ((pPrefix = 0) AND (LenPrefix>0)) OR
   ((pSuffix = 0) AND (LenSuffix>0)) THEN
	Error := COMERROR_INVALIDPOINTER;
	state := 0;
	RETURN;
END_IF

IF state = 0 THEN
	DataReceived := FALSE;
	busy := FALSE;
	Error := 0;
	RxTimeout := FALSE;
	LenReceiveData := 0;
	l := 0;
	state := 1;
ELSE
	REPEAT
		(* receive one character *)
		Receive(RXbuffer:=RXbuffer);

		TimeoutTimer( IN:=Receive.ByteReceived, PT:=iTimeout );

		IF  Receive.ByteReceived THEN
			c := Receive.ReceivedByte;
			IF state = 1 THEN
				busy := TRUE;
				l := 0;
				ptrPrefix := pPrefix;
				pData := pReceiveData;
				iTimeout := Timeout;
				IF LenPrefix > 0 THEN
					state := 10;
				ELSIF LenSuffix > 0 THEN
					state := 20; (* wait for suffix *)
				ELSE
					state := 30; (* wait until data size reached *)
				END_IF
			END_IF

			CASE state OF
				10 :	(* Wait for prefix *)
					IF l >= SizeReceiveData THEN
						(* size of data block reached *)
						Error := COMERROR_DATASIZEOVERRUN;
						DataReceived := TRUE;
						LenReceiveData := l;
						busy := FALSE;
						state := 0;
					ELSE
						l := l + 1;
						pData^ := c;
						IF l <= LenPrefix THEN
							IF ptrPrefix^ <> pData^ THEN
								l := 0;
							ELSE
								IF l = LenPrefix THEN
									IF LenSuffix > 0 THEN
										state := 20; (* wait for suffix *)
									ELSE
										state := 30; (* wait until data size reached *)
									END_IF
								END_IF
							END_IF
						END_IF
						(* pData := _AddPointer(ReceivedData, l); *)
						pw := pReceiveData;
						pw := pw + l;
						pData := pw;
						(* ptrPrefix := _AddPointer(Prefix, l); *)
						pw := pPrefix;
						pw := pw + l;
						ptrPrefix := pw;
					END_IF

				20 : (* Wait for suffix *)
					IF l >= SizeReceiveData THEN
						(* size of data block reached *)
						Error := COMERROR_DATASIZEOVERRUN;
						DataReceived := TRUE;
						LenReceiveData := l;
						busy := FALSE;
						state := 0;
					ELSE
						l := l + 1;
						pData^ := c;
						(* pData := ReceivedData +  l; *)
						pw := pReceiveData; pw := pw + l; pData := pw;
						IF (LenSuffix > 0) AND (l >= LenPrefix + LenSuffix) THEN
							p1 := pData;
							(* p2 := Suffix + LenSuffix; *)
							pw := pSuffix; pw := pw + LenSuffix;	p2 := pw;
							isEqual := TRUE;
							FOR i := 1 TO LenSuffix DO
								(* p1 := p1 - 1; *)
								pw := p1; pw := pw - 1; p1 := pw;
								(* p2 := p2 - 1; *)
								pw := p2; pw := pw - 1; p2 := pw;
								IF p1^ <> p2^ THEN
									isEqual := FALSE;
									EXIT;
								END_IF
							END_FOR
							IF isEqual THEN
								DataReceived := TRUE;
								LenReceiveData := l;
								busy := FALSE;
								state := 0;
							END_IF
						END_IF
					END_IF

				30 : (* receive until size of data block reached *)
					l := l + 1;
					pData^ := c;
					(* pData := ReceivedData +  l; *)
					pw := pReceiveData; pw := pw + l; pData := pw;
					IF l >= SizeReceiveData THEN
						(* size of data block reached *)
						DataReceived := TRUE;
						LenReceiveData := l;
						busy := FALSE;
						state := 0;
					END_IF
			END_CASE
		ELSE
			(* no char received *)
			IF state > 1 AND l > 0 AND iTimeout > T#0s AND NOT TimeoutTimer.Q THEN
				DataReceived := TRUE;
				LenReceiveData := l;
				busy := FALSE;
				RxTimeout := TRUE;
				state := 0;
			END_IF
		END_IF
	UNTIL NOT busy OR NOT Receive.ByteReceived
	END_REPEAT
END_IF

END_FUNCTION_BLOCK

// POUs/COMlibV2/Send + Receive/ReceiveString
FUNCTION_BLOCK ReceiveString
VAR_INPUT
	Prefix 			: STRING;
	Suffix 			: STRING;
	Timeout			: TIME;
	Reset  			: BOOL;
END_VAR
VAR_OUTPUT
	StringReceived	: BOOL;
	Busy 			: BOOL;
	Error			: ComError_t;
	RxTimeout 		: BOOL;
END_VAR
VAR_IN_OUT
	ReceivedString 	: STRING;
	RXbuffer 			: COMbuffer;
END_VAR
VAR
	ReceiveStringStandard: _ReceiveString;
	ErrorCountPrefix 		: INT; (* invalid characters received before prefix *)
	ReceivedPrefix 		: STRING;(* received prefix including invalid characters *)
END_VAR

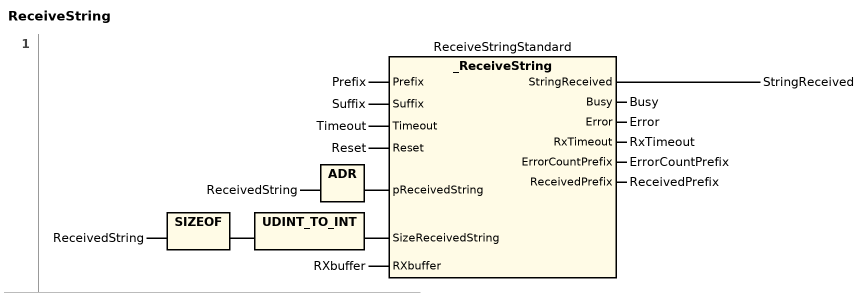
// NETWORK 1
ReceiveStringStandard(
    Prefix := Prefix,
    Suffix := Suffix,
    Timeout := Timeout,
    Reset := Reset,
    pReceivedString := ADR(ReceivedString),
    SizeReceivedString := UDINT_TO_INT(SIZEOF(ReceivedString)),
    RXbuffer := RXbuffer,
    Busy => Busy,
    Error => Error,
    RxTimeout => RxTimeout,
    ErrorCountPrefix => ErrorCountPrefix,
    ReceivedPrefix => ReceivedPrefix); // _ReceiveString
StringReceived := ReceiveStringStandard.StringReceived;

END_FUNCTION_BLOCK

// POUs/COMlibV2/Send + Receive/ReceiveString255
FUNCTION_BLOCK ReceiveString255
VAR_INPUT
	Prefix 			: STRING;
	Suffix 			: STRING;
	Timeout			: TIME;
	Reset  			: BOOL;
END_VAR
VAR_OUTPUT
	StringReceived	: BOOL;
	Busy 			: BOOL;
	Error			: ComError_t;
	RxTimeout 		: BOOL;
END_VAR
VAR_IN_OUT
	ReceivedString 	: STRING(255);
	RXbuffer 			: COMbuffer;
END_VAR
VAR
	ReceiveStringStandard: _ReceiveString;
	ErrorCountPrefix : INT; (* invalid characters received before prefix *)
	ReceivedPrefix : STRING;(* received prefix including invalid characters *)
END_VAR

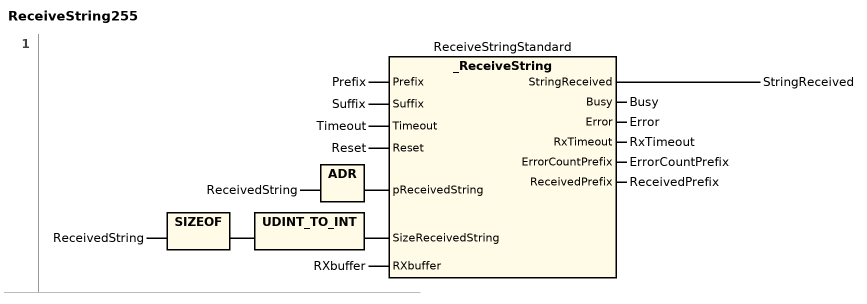
// NETWORK 1
ReceiveStringStandard(
    Prefix := Prefix,
    Suffix := Suffix,
    Timeout := Timeout,
    Reset := Reset,
    pReceivedString := ADR(ReceivedString),
    SizeReceivedString := UDINT_TO_INT(SIZEOF(ReceivedString)),
    RXbuffer := RXbuffer,
    Busy => Busy,
    Error => Error,
    RxTimeout => RxTimeout,
    ErrorCountPrefix => ErrorCountPrefix,
    ReceivedPrefix => ReceivedPrefix); // _ReceiveString
StringReceived := ReceiveStringStandard.StringReceived;

END_FUNCTION_BLOCK

// POUs/COMlibV2/Send + Receive/SendData
FUNCTION_BLOCK SendData
VAR_INPUT
	pSendData 	: POINTER TO BYTE;
	Length 		:  UDINT;
END_VAR
VAR_OUTPUT
	Busy 		: BOOL;
	Error		: ComError_t;
END_VAR
VAR_IN_OUT
	TXbuffer		: COMbuffer;
END_VAR
VAR
	pos : UINT;
	Send : SendByte;
	c : BYTE;
	dp : POINTER TO BYTE;
	dpw : XWORD;
END_VAR

	IF NOT Busy THEN
		pos := 1;
		dp := pSendData;
		Busy := TRUE;
		IF dp = 0 THEN
			error := COMERROR_INVALIDPOINTER;
			busy := FALSE;
			RETURN;
		END_IF
	END_IF

	IF Send.Busy THEN
		Send( TxBuffer := TxBuffer );
		Error := Send.Error; (* 2011-06-24 JANZ: line added because otherwise in case of buffer overrun at last byte: error keeps at output although it was sent successfully. *)
	ELSE
		REPEAT
(*			IF NOT Send.Busy OR Send.Error = COMERROR_TXBUFFOVERRUN THEN	*)	(* 2011-01-19 JANZ if condition removed because line is needless (Send.Busy always FALSE here) *)
				IF pos > Length THEN
					busy := FALSE;
				ELSE
					c := dp^;
					Send( SendByte := c, TxBuffer := TxBuffer );
					Error := Send.Error;
(*					IF Send.Error = 0 THEN	 *)	(* 2010-02-19 KSt IF condition removed *)
					pos := pos + 1;
					(* increment pointer *)
					dpw := dp;
					dpw := dpw + 1;
					dp := dpw;
(*					END_IF; *)					(* 2010-02-19 KSt IF condition removed *)
				END_IF
(*			END_IF	*)							(* 2011-01-19 JANZ if condition removed *)
		UNTIL Send.Busy OR NOT busy
		END_REPEAT
	END_IF

END_FUNCTION_BLOCK

// POUs/COMlibV2/Send + Receive/SendString255
FUNCTION_BLOCK SendString255
VAR_INPUT
	SendString:	STRING(255);
END_VAR
VAR_OUTPUT
	Busy : 		BOOL;
	Error:		ComError_t;
END_VAR
VAR_IN_OUT
	TXbuffer:	COMbuffer;
END_VAR
VAR
END_VAR
VAR
	SendStringStandard: _SendString;
END_VAR

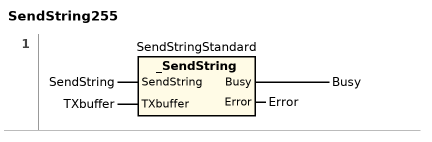
// NETWORK 1
SendStringStandard(SendString := SendString, TXbuffer := TXbuffer, Error => Error); // _SendString
Busy := SendStringStandard.Busy;

END_FUNCTION_BLOCK

// POUs/COMlibV2/Version/Get_ComLib_Version
FUNCTION Get_ComLib_Version : STRING(20)
VAR_INPUT
	bGet : BOOL;
END_VAR
(* Version history:
Date[DD.MM.YYYY]| Version	| created under	| Author|	Remark
----------------------------------------------------------------------------------------------------
07.07.2000		| 1.004.000	|				| KSt	|	version tracking 
15.11.2000		| 1.005.000	|				| KSt	|	initialization revised
31.08.2001		| 1.005.001	|				| KSt	|	STRING(255) with ComLib255 for ReceiveString and SendString
29.11.2001		| 1.005.002	|				| KSt	|	receive of null byte checked in ReceiveString
20.12.2001		| 1.006.000	|				| KSt	|	new FB ReceiveData, SendData, ReceiveString255 and SendString255
24.05.2002		| 1.006.002	|				| KSt	|	comments in KL6Config changed
03.06.2002		| 1.007.000	|				| KSt	|	string copy routine in receive string changed
30.12.2002		| 1.007.002	|				| KSt	|	check if input parameters have changed in ReceiveString
22.12.2004		| 2.000.000	|				| KSt	|	universal hardware independent background communication (SerialLineControl)
														universal hardware independent KL6 configuration for all KL6 types (KL6configuruation)
														register access to all KL6 types (KL6WriteRegisters)
01.03.2005		| 2.000.001	|				| KSt	|	universal hardware independent reset block ComReset for all KL6 terminals 
29.04.2005		| 2.000.002	|				| KSt	|	fix in SendString and SendData for corret buffer full handling 
18.10.2005 		| 2.000.003	|				| KSt	|	kein Zurücksetzen des ContinousModeStart bits solange noch weitere Daten anstehen
17.07.2006 		| 2.000.004	|				| KSt	|	fix in CHR to avoid CX9000 stack an initialization issue
25.04.2007 		| 2.000.005	|				| KSt	|	error message with KL6xxx 3 byte alternative mode terminals at BC couplers
20.05.2008		| 2.000.006	|				| KSt	|	_SendString modified. LEN is now calculated out of the REPEAT loop;
														data type for EL6001 added (compatibel to KL6 22B)
01.08.2008		| 2.001.000	|				| KSt	|	IP6002-0001 with 11 data bytes supported
07.09.2009		| 2.002.000	|				| KSt	|	M8000 modules supported
15.09.2009		| 2.002.001	|				| KSt	|	data types adapted to PlcControl V3 (INT->UINT etc.)
19.02.2010 		| 2.002.003	|				| KSt	|	SendData and SendString : buffer overrun issue fixed
04.08.2010		| 2.003.000	| v2.11 R2(2013)| JANZ	|	TcAdsSerialCommServer supported (virtual serial COM ports supported) [beta version]
12.01.2011		| 2.003.001	|				| KSt	|	less important fix in _strncpy
19.05.2011		| 2.003.002	| v2.11 R2(2030)| JANZ	|	FB_ASC_SerialLineControl: interface and behaivor updated (behaivor also improved if serial port is already or not yet opened);
														SendData: optimized: needless if-condition removed; folder structure in library updated
06.07.2011		| 2.003.003	| v2.11 R2(2030)| JANZ	|	FB_ASC_SerialLineControl: enum types used in input structure; Delay of 100ms added after win32 error occurred; TraceLevel updated
14.07.2011		| 2.003.004	| v2.11 R2(2030)| JANZ	|	all prefixes removed at new objects [still beta version]
24.08.2011		| 2.003.005	| v2.11 R2(2036)| KSt	|	Baudrate 300 and 600 added to KL6configuration - early reset of reset flag in KL6configuration
12.09.2011		| 2.003.006	| v2.11 R2(2036)| KSt	|	KL6configuration: check of register access bit avoids wrong feedback of reset bit if register communication is still active
13.11.2011		| 2.003.007	| v2.11 R2(2040)| JANZ	|	SerialLineControlAds: error codes (RD_FAILURE and WR_FAILURE) added
10.04.2012		| 2.003.008	| v2.11 R3(2217)| JANZ	|	release of new ads functionality; folder structure of library improved
*)

Get_ComLib_Version := VERSION_COMLIB;

END_FUNCTION

// POUs/COMlibV2/ComReset
(*=================================================================
 *	ComReset
 *	The function block resets all kinds of KL6 terminals.
 *	The terminal internal receive and transmit buffers are cleared.
 *=================================================================
 *)
FUNCTION_BLOCK ComReset
VAR_INPUT
	Execute	: BOOL;
	pComIn		: POINTER TO ARRAY[0..65] OF BYTE;	(* pointer to any KL6 or COM-Port process image *)
	pComOut	: POINTER TO ARRAY[0..65] OF BYTE;	(* pointer to any KL6 or COM-Port process image *)
	SizeComIn	:	UINT;
END_VAR
VAR_OUTPUT
	Done		: 	BOOL;
	Busy		:	BOOL;
	Error		: 	BOOL;
	ErrorID		:	ComError_t;
END_VAR
VAR CONSTANT
	TIME_OUT_VALUE	: TIME  := T#100MS;
	RESETMASK_STANDARD		: WORD := 2#00000100;
	RESETMASK_ALTERNATIVE	: WORD := 2#00000100_00000000;
END_VAR
VAR
	Timeout: TON;
	state: INT;
	pCTRL: POINTER TO WORD;
	pSTATUS: POINTER TO WORD;
	ResetMask : WORD;
	TriggerExecute: R_TRIG;
END_VAR

TriggerExecute(CLK:=Execute);
CASE state OF
	0 : (* init *)
		Busy := FALSE;
		IF NOT Execute THEN
			Done := FALSE;
		END_IF
		IF TriggerExecute.Q THEN
			IF pComIn=0 OR pComOut=0 THEN
				Error := TRUE;
				ErrorID := COMERROR_INVALIDPOINTER;
			ELSE
				Done := FALSE;
				Error := FALSE;
				ErrorID := 0;
				pCTRL := pComOut;
				pSTATUS := pComIn;
				(* size=5 then KL6/3Byte/Alternative-Mode else Standard-Mode *)
				ResetMask := SEL(SizeComIn=5, RESETMASK_STANDARD, RESETMASK_ALTERNATIVE);
				Timeout(IN:=FALSE);
				Busy := TRUE;
				pCTRL^ := ResetMask;
				state := state + 1;
			END_IF
		END_IF

	1:	(* reset terminal *)
		pCTRL^ := ResetMask;
		Timeout(IN:=TRUE , PT:=TIME_OUT_VALUE );
		IF  ( pSTATUS^ AND ResetMask) <> 0 THEN
			Timeout(IN:=FALSE);
			pCTRL^ := pCTRL^ AND NOT RESETMASK;
  			state := state + 1;
		ELSIF Timeout.Q THEN
			Error := TRUE;
			ErrorID := COMERROR_TIMEOUT;
			pCTRL^ := pCTRL^ AND NOT RESETMASK;
			state := 0;
		END_IF

	2:	(* end reset terminal *)
		pCTRL^ := pCTRL^ AND NOT RESETMASK;
		Timeout(IN:=TRUE , PT:=TIME_OUT_VALUE );
		IF  ( pSTATUS^ AND ResetMask) = 0 THEN
			Timeout(IN:=FALSE);
			Done := TRUE;
  			state := 0;
		ELSIF Timeout.Q THEN
			Error := TRUE;
			ErrorID := COMERROR_TIMEOUT;
			state := 0;
		END_IF

END_CASE

IF state=0 THEN
	Busy := FALSE;
END_IF

END_FUNCTION_BLOCK

// POUs/COMlibV2/ClearComBuffer
(*=================================================================
 *	
 *	Modul:	ClearComBuffer
 *  			The function block clears the software read/write
 *			buffer but it will not clear data buffers inside the
 *			hardware e. g. KL-6xxx.
 *	Date:	01.12.1998
 *
 *=================================================================
 *)
FUNCTION_BLOCK ClearComBuffer
VAR_INPUT
END_VAR
VAR_OUTPUT
END_VAR
VAR_IN_OUT
	Buffer :		COMbuffer;
END_VAR
VAR
END_VAR

	Buffer.blocked := TRUE;	(* block fast PLC Task *)
	Buffer.Count := 0;
	Buffer.FreeByte := SIZEOF(Buffer.Buffer) - Buffer.Count;
	Buffer.RdIdx := 0;
	Buffer.WrIdx := 0;
	Buffer.blocked := FALSE;	(* unblock fast PLC Task *)

END_FUNCTION_BLOCK
